IF NOT bOpenClose THEN
	eOpClCtrl := eCtrl;
	THIS^.bCloseWithPiece := bCloseWithPiece;
	fbList.A_AddHeadValue(hList := hList, putValue:= E_Action.ACTION_OpenClose);
	bOpenClose := TRUE;
ELSE
	RETURN;
END_IF

bBusy := TRUE;
eCurrentState := E_MachineState.MACHINESTATE_Active;
END_METHOD

METHOD M_SetAllProps : ERRORID
VAR_INPUT
	refCmdData : REFERENCE TO  ST_CmdData;
END_VAR

VAR
	
END_VAR
M_SetAllProps := SUPER^.M_SetAllProps(refCmdData);

IF M_SetAllProps > 0 THEN
	RETURN;
END_IF

pGripperRef := ADR(pFbMultiZ^.aFbGripperRef[pZAxisRef^.nChannel]);
pZAxisRef^.eFixedToolType := E_MzToolType.TOOL_TYPE_Gripper;
END_METHOD

PROPERTY P_bVialDetector : BOOL
GET
P_bVialDetector :=  pGripperRef^.P_bVialDetector;
END_GET
END_PROPERTY

PROPERTY P_eCurrentGripperState : E_GripperState
GET
P_eCurrentGripperState := pGripperRef^.P_eGripperState;
END_GET
END_PROPERTY

END_FUNCTION_BLOCK

// ---- Objects/Targets/Active/FB_PowderStation.TcPOU
FUNCTION_BLOCK FB_PowderStation EXTENDS FB_ActiveTarget IMPLEMENTS I_SlotTarget
VAR
	
	nNoOfSpecPoints 	: USINT;
	stPickPoint			: ST_3DPoint;
	nLevelOffset		: DINT;
	
	nNoOfSlots			: USINT;
	fbVialSlot			: FB_PieceSlot(pOwner:= THIS);


	//Hardware-Verküpfung
	pPowdStatRef		: POINTER TO FB_HwRefPowderStat;
	
	//Variablen allgemeine Statemachine
	fbSdoWrite			: FB_SDO_WRITE;
	
	//****************************************Aktionvariablen****************************************************
	bActionLock			: ARRAY[50..150] OF BOOL;

	//Action: "Shaking"	(Rüttelmotor schalten)
	bShaking			: BOOL;
	nStateA_Shaking		: USINT;
	nVibrationPower1	: UINT;
	nVibrationPower2	: UINT;
	nVibrationPower3	: UINT;

	//Action: "Leveling"	(Pulver rütteln und auf Höhe bringen)
	bLeveling			: BOOL;				//Action A_Leveling() aktiv setzen
	nStateA_Leveling	: USINT;			//State von A_Leveling()
	tShakingTime		: TIME;
	timer				: TON;
	
	//Action: "Reload"	(Stößel in untere Position fahren zum nachfüllen)
	bReload				: BOOL;
	nStateA_Reload		: USINT;
	
	//Action: "TakePicture"
	bTakePicture			: BOOL;
	nStateA_TakePicture		: USINT;
	tDelayTakePicture		: TIME;
	timerTakePicture		: TON;
	nRequestArg1			: DINT;
	nRequestArg2			: DINT;	
	
END_VAR

IF bInitFB THEN
	bInitFB := FALSE;
	F_CreateLinkedListHnd( ADR( aNodes ), SIZEOF( aNodes ), hList );
	//Fehlerstruktur vorausfüllen
	stError.ObjectId := nObjectID;
	stError.HardwareGrp := E_HardwareGrp.Nothing;
	stError.POU := E_POU.POU_FB_PowderStation;
END_IF

CASE eCurrentState OF
	E_MachineState.MACHINESTATE_Active:
		//BasicActions ausführen
		IF bInit THEN	//Initialisieren
			A_Init();
			IF nStateA_Init >= 80 THEN
				IF nStateA_Init >= 99 THEN
					bError := TRUE;
				END_IF
				bInit := FALSE;
				nStateA_Init := 0;
				M_RemoveListEntry(nSearchValue:= E_Action.ACTION_Init);
			END_IF
		END_IF

		IF bShaking THEN
			A_Shaking();
			IF nStateA_Shaking >= 80 THEN
				IF nStateA_Shaking >= 99 THEN
					bError := TRUE;
				END_IF
				bShaking := FALSE;
				nStateA_Shaking := 0;
				M_RemoveListEntry(nSearchValue:= E_Action.ACTION_PowdStatShaking);
			END_IF
		END_IF
		
		IF bLeveling THEN
			A_Leveling();
			IF nStateA_Leveling >= 80 THEN
				IF nStateA_Leveling >= 99 THEN
					bError := TRUE;
				END_IF
				bLeveling := FALSE;
				nStateA_Leveling := 0;
				M_RemoveListEntry(nSearchValue:= E_Action.ACTION_PowdStatLeveling);
			END_IF
		END_IF
		
		IF bReload THEN
			A_Reload();
			IF nStateA_Reload >= 80 THEN
				IF nStateA_Reload >= 99 THEN
					bError := TRUE;	
				END_IF
				bReload := FALSE;
				nStateA_Reload := 0;
				M_RemoveListEntry(nSearchValue:= E_Action.ACTION_PowdStatReload);
			END_IF
		END_IF

		IF bTakePicture THEN
			A_TakePicture();
			IF nStateA_TakePicture >= 80 THEN
				IF nStateA_TakePicture >= 99 THEN
					bError := TRUE;	
				END_IF
				bTakePicture := FALSE;
				nStateA_TakePicture := 0;
				M_RemoveListEntry(nSearchValue:= E_Action.ACTION_TakePicture);
			END_IF
		END_IF		
		
		IF bStop THEN	//alle Actions stoppen
			A_Stop();
			IF nStateA_Stop >= 80 THEN
				IF nStateA_Stop >= 99 THEN
					bError := TRUE;
				END_IF
				bStop := FALSE;
				nStateA_Stop := 0;
				bCanceled := TRUE;
				M_RemoveListEntry(nSearchValue:= E_Action.ACTION_Stop);
			END_IF							
		END_IF

		IF hList.nCount = 0 THEN
			eCurrentState := E_MachineState.MACHINESTATE_Ready;
		END_IF

		IF bError  THEN
			eCurrentState := E_MachineState.MACHINESTATE_Error;
		END_IF

	E_MachineState.MACHINESTATE_Reset:
		A_Reset();
		IF nStateA_Reset = 80 THEN
			nStateA_Init := 0;
			nStateA_Stop := 0;
			nStateA_Reset := 0;
			bBusy := FALSE;
			bError := FALSE;
			bStopAllOnError := FALSE;
			fbList.A_Reset( hList := hList);
			MEMSET(ADR(bActionLock),0,SIZEOF(bActionLock));
			nErrorId := 0;
			stError.Cmd := 0;
			stError.ErrorId := 0;
			eCurrentState := E_MachineState.MACHINESTATE_Idle;
		ELSIF
			nStateA_Reset = 99 THEN
			fbErrorList.M_Add(stError);
			nStateA_Reset := 0;
			bBusy := FALSE;
			bError := TRUE;
			eCurrentState := E_MachineState.MACHINESTATE_Error;			
		END_IF
	
	E_MachineState.MACHINESTATE_Ready:
		bBusy := FALSE;
		eCurrentState := E_MachineState.MACHINESTATE_Idle;
	
	E_MachineState.MACHINESTATE_Error:
		bBusy := FALSE;
END_CASE

//Prozessdaten aktualisieren
stProcessData.nObjId := nObjectID;
stProcessData.n32Data[0] := BOOL_TO_DINT(bIsInit);
stProcessData.n32Data[1] := eCurrentState;
stProcessData.n32Data[2] := stError.ErrorId;
stProcessData.n32Data[3] := BOOL_TO_DINT(pPowdStatRef^.bLevelOk);	
stProcessData.n32Data[4] := BOOL_TO_DINT(pPowdStatRef^.bLevelLow);
stProcessData.n32Data[5] := BOOL_TO_DINT(pPowdStatRef^.bOnReloadPos);
stProcessData.n32Data[6] := BOOL_TO_DINT(pPowdStatRef^.bVibrationIsOn);
//stProcessData.n32Data[7] := BOOL_TO_DINT(pPowdStatRef^.bCoverIsClosed);
stProcessData.n32Data[7] := BOOL_TO_DINT(pPowdStatRef^.bVialSensor);
stProcessData.n32Data[8] := BOOL_TO_DINT(pPowdStatRef^.bLevelSensor);
stProcessData.n32Data[9] := BOOL_TO_DINT(pPowdStatRef^.bHeaterIsOn);

stProcessData.n32Data[10] := pPowdStatRef^.nTempActual;
IF pPowdStatRef^.P_nCameraLight > 0 THEN
	stProcessData.n32Data[11] := 1;
ELSE
	stProcessData.n32Data[11] := 0;
END_IF
aObjProcData[nNotifyId] := stProcessData;

ACTION A_Init:
CASE nStateA_Init OF
	0:	//Wenn in Error, dann Error zurücksetzen
		bIsInit := FALSE;
		pPowdStatRef^.P_bStartLeveling := FALSE;
		pPowdStatRef^.P_bStartReload := FALSE;
		pPowdStatRef^.P_bVibrationOn := FALSE;
		IF pPowdStatRef^.bErr THEN
			pPowdStatRef^.P_bResetError := TRUE;
			nStateA_Init := 1;
		ELSE
			nStateA_Init := 2;
		END_IF

	1:	//Warten bis Error zurückgesetzt	
		IF NOT pPowdStatRef^.bErr THEN
			pPowdStatRef^.P_bResetError := FALSE;
			nStateA_Init := 2;
		END_IF
		
	2:	//Stöße in ReladPos fahren, wenn noch nicht geschehen
		IF NOT pPowdStatRef^.bOnReloadPos THEN
			pPowdStatRef^.P_bStartReload := TRUE;
			nStateA_Init := 3;
		ELSE
			nStateA_Init := 80;
			bIsInit := TRUE;
		END_IF
	
	3:	//Warten bis Stößel in ReloadPos
		IF pPowdStatRef^.bOnReloadPos THEN
			pPowdStatRef^.P_bStartReload := FALSE;
			nStateA_Init := 80;
			bIsInit := TRUE;	
		END_IF
		IF pPowdStatRef^.bError THEN
			stError.ErrorId := E_ErrorIdCmd.ERRORID_DeviceInErrorState;
			stError.POUState := nStateA_Init;
			nStateA_Init := 99;		
		END_IF
	
	70:	//Initialisierung abbrechen
		pPowdStatRef^.P_bResetError := FALSE;	
		pPowdStatRef^.P_bStartReload := FALSE;
		nStateA_Init := 80;
	
END_CASE

//Errorhandling
IF nStateA_Init = 99 THEN
	stError.Cmd := E_Action.ACTION_Init;
	stError.POUAction := E_POUACT.POUACT_A_Init;
	fbErrorList.M_Add(stError);
END_IF
END_ACTION

ACTION A_Leveling:
stError.POUState := nStateA_Leveling;

IF pPowdStatRef^.bError THEN
	stError.ErrorId := pPowdStatRef^.nError;
	nStateA_Leveling := 99;
	pPowdStatRef^.P_bVibrationOn := FALSE;
END_IF

CASE nStateA_Leveling OF
	0:	//LevelOffset schreiben
		fbSdoWrite(sAdsNetID:= pPowdStatRef^.P_sAdsNetId, nPortNr:= pPowdStatRef^.P_nAdsPort, nIndex:= 16#2104,
					nSubIndex:= 0, nDataLength:= 2, nData:= ABS(nLevelOffset), bExecute:= TRUE);
		IF NOT fbSdoWrite.bBusy THEN
			IF fbSdoWrite.bError THEN
				stError.ErrorId := fbSdoWrite.nAdsErrorId;
				nStateA_Leveling := 99;
			ELSE
				pPowdStatRef^.P_bStartReload := TRUE;
				nStateA_Leveling := 1;
			END_IF
			fbSdoWrite(bExecute:= FALSE);
		END_IF

	1:	//OnReloadPos?
		//Timeout
		timer(IN:=TRUE, PT:= T#5S);
		IF timer.Q THEN
			timer(IN:= FALSE);
			stError.ErrorId := E_ErrorIdCmd.ERRORID_TimeOut;
			nStateA_Leveling := 99;
		END_IF
 
		IF pPowdStatRef^.bOnReloadPos THEN
			timer(IN:=FALSE);
			pPowdStatRef^.P_bStartReload := FALSE;
			IF pPowdStatRef^.bLevelSensor THEN
				stError.ErrorId := E_ErrorIdCmd.ERRORID_PowdDetectOnReloadPos;
				nStateA_Leveling := 99;				
			ELSE
				//ShakerOn, Start Timer
				pPowdStatRef^.P_bVibrationOn := TRUE;
				timer(IN:=TRUE, PT:= tShakingTime);
				nStateA_Leveling := 2;
			END_IF
		END_IF
		
	2:	//Warten bis Timer abgelaufen
		timer();
		IF timer.Q THEN
			timer(IN:= FALSE);
			pPowdStatRef^.P_bVibrationOn := FALSE;
			pPowdStatRef^.P_bStartLeveling := TRUE;
			nStateA_Leveling := 3;
		END_IF
		
	3:	//Warten bis Leveling fertig
		IF pPowdStatRef^.bLevelOk THEN
			pPowdStatRef^.P_bStartLeveling := FALSE;
			nStateA_Leveling := 80;
		ELSIF pPowdStatRef^.bLevelLow THEN
			pPowdStatRef^.P_bStartLeveling := FALSE;
			stError.ErrorId := E_ErrorIdCmd.ERRORID_PowdLevelLow;
			nStateA_Leveling := 99;
		END_IF
		
	70:	//Abbrechen
		pPowdStatRef^.P_bVibrationOn := FALSE;
		pPowdStatRef^.P_bStartLeveling := FALSE;
		pPowdStatRef^.P_bStartReload := FALSE;
		timer(IN:= FALSE);
		nStateA_Leveling := 80;
END_CASE

//Errorhandling
IF nStateA_Leveling = 99 THEN
	stError.Cmd := E_Action.ACTION_PowdStatLeveling;
	stError.POUAction := E_POUACT.POUACT_A_Leveling;
	fbErrorList.M_Add(stError);
END_IF
END_ACTION

ACTION A_Reload:
IF pPowdStatRef^.nError > 0 OR pPowdStatRef^.bError THEN
	stError.POUState := nStateA_Reload;
	stError.ErrorId := pPowdStatRef^.nError;
	nStateA_Reload := 99;
END_IF

CASE nStateA_Reload OF
	0:
		pPowdStatRef^.P_bStartReload := TRUE;
		nStateA_Reload := 1;
		
	1:	//Warten bis Stößel in ReloadPos
		IF pPowdStatRef^.bOnReloadPos THEN
			pPowdStatRef^.P_bStartReload := FALSE;
			nStateA_Reload := 80;
		END_IF
		
	70:	//Abbrechen
		pPowdStatRef^.P_bStartReload := FALSE;
		nStateA_Reload := 80;
END_CASE

//Errorhandling
IF nStateA_Reload = 99 THEN
	stError.Cmd := E_Action.ACTION_PowdStatShaking;
	stError.POUAction := E_POUACT.POUACT_A_Shaking;
	fbErrorList.M_Add(stError);
END_IF
END_ACTION

ACTION A_Reset:
CASE nStateA_Reset OF
	0:
		nStateA_Reset := 80;
END_CASE
END_ACTION

ACTION A_Shaking:
CASE nStateA_Shaking OF
	0:	
		pPowdStatRef^.P_bVibrationOn := TRUE;
		IF tShakingTime > T#0MS THEN
			timer(IN:= TRUE, PT:= tShakingTime);
			nStateA_Shaking := 1;
		END_IF
	1:
		timer();
		IF timer.Q THEN
			pPowdStatRef^.P_bVibrationOn := FALSE;
			timer(IN:= FALSE);
			nStateA_Shaking := 80;
		END_IF
		
	70:	//Abrechen
		pPowdStatRef^.P_bVibrationOn := FALSE;
		timer(IN:=FALSE);
		nStateA_Shaking := 80;
END_CASE
END_ACTION

ACTION A_Stop:
CASE nStateA_Stop OF
	0:
		IF nStateA_Init < 70 AND bInit THEN	//Initialisieren abbrechen
			nStateA_Init := 70;
			nStateA_Stop := 1;	
		END_IF
		
		IF nStateA_Leveling < 70 AND bLeveling THEN
			nStateA_Leveling := 70;
			nStateA_Stop := 1;
		END_IF
		
		IF nStateA_Shaking < 70 AND bShaking THEN
			nStateA_Shaking := 70;
			nStateA_Stop := 1;
		END_IF
		
		IF nStateA_Reload < 70 AND bReload THEN
			nStateA_Reload := 70;
			nStateA_Stop := 1;
		END_IF

	1:	//Warten bis alle Actions fertig abgebrochen
		IF hList.nCount = 1 THEN	//nur der Eintrag von Stop
			nStateA_Stop := 80;
		END_IF
END_CASE
END_ACTION

ACTION A_TakePicture:
IF nStateA_TakePicture = 0 THEN //Timer starten
	timerTakePicture(IN:= TRUE, PT:= tDelayTakePicture);
	IF timerTakePicture.Q THEN
		timerTakePicture(IN:= FALSE);
		stInterResponse.eInteractMessageType := E_InteractMessageType.INTERACTMES_NONE;
		stInteractRequest.eInteractMessageType := E_InteractMessageType.INTERACTMES_WaitForUser;
		stInteractRequest.nObjectId := nObjectID;
		stInteractRequest.nArg1 := nRequestArg1;
		stInteractRequest.nArg2 := nRequestArg2;
		nStateA_TakePicture := 1;
	END_IF
ELSIF nStateA_TakePicture = 1 THEN //Auf InteractResponse warten
	IF stInterResponse.eInteractMessageType = E_InteractMessageType.INTERACTMES_Continue OR 
							stInterResponse.eInteractMessageType = E_InteractMessageType.INTERACTMES_Cancel THEN
		stInteractRequest.eInteractMessageType := E_InteractMessageType.INTERACTMES_NONE;
		nStateA_TakePicture := 80;
	END_IF
ELSIF nStateA_TakePicture = 70 THEN //Abbrechen
	timerTakePicture(IN:= FALSE);
	stInteractRequest.eInteractMessageType := E_InteractMessageType.INTERACTMES_NONE;
	nStateA_TakePicture := 80;
END_IF
END_ACTION

METHOD FB_init : BOOL
VAR_INPUT
	bInitRetains : BOOL; // if TRUE, the retain variables are initialized (warm start / cold start)
	bInCopyCode : BOOL;  // if TRUE, the instance afterwards gets moved into the copy code (online change)
END_VAR
eObjectType := E_ObjectType.OBJECTTYPE_PowderStation;
eObjectGroup := E_ObjectGroup.OBJECTGROUP_Target OR E_ObjectGroup.OBJECTGROUP_Device;
END_METHOD

METHOD M_AddChild : ERRORID
VAR_INPUT
	pObject : POINTER TO FB_Object;
	nSlotNr	: UINT;
	nIndex 	: INT;	
END_VAR
IF pObject > 0 THEN
	IF nSlotNr = fbVialSlot.P_nNr THEN //Reactor besitzt nur den VialSlot
		IF fbVialSlot.P_pChild = 0 THEN
			//Object darf selber noch an keinem Parent hängen
			IF pObject^.P_pParentObject = 0 THEN
				fbVialSlot.P_pChild := pObject;
				pObject^.P_pObjCollectNode := pObjCollectNode^.nodes.M_AddNewNode(pObject,nIndex);
				pObject^.M_UpdateParent();
			ELSE
				M_AddChild := E_ErrorIdObjMgmt.ERRORID_ObjectAlreadyOnAnotherParent;
			END_IF
		ELSE //Slot bereits belegt
			M_AddChild := E_ErrorIdObjMgmt.ERRORID_SlotIsAlreadyOccupied;
		END_IF		
	ELSE
		M_AddChild := SUPER^.M_AddChild(pObject,nSlotNr,nIndex);
	END_IF
ELSE
	M_AddChild := E_ErrorIdObjMgmt.ERRORID_InvalidParentObject;
END_IF
END_METHOD

METHOD M_ApplyPos : ERRORID
VAR_INPUT
	eTargetRef 		: E_TargetRef;
	nPointSlotNr	: UINT;
	stPos 			: ST_3DPoint;
	bXPos			: BOOL;
	bYPos			: BOOL;
	bZPos			: BOOL;	
END_VAR

VAR
	stAbsPos		: ST_3DPoint;
END_VAR
IF eTargetRef = E_TargetRef.TARGETREF_SpecPoint THEN
	IF nPointSlotNr = 1 THEN
		stAbsPos := P_stAbsPosLB;
		IF bXPos THEN
			stPickPoint.X := stPos.X - stAbsPos.X;	
		END_IF
		IF bYPos THEN
			stPickPoint.Y := stPos.Y - stAbsPos.Y;	
		END_IF
		IF bZPos THEN
			stPickPoint.Z := stPos.Z - stAbsPos.Z;	
		END_IF
	ELSE
		M_ApplyPos := E_ErrorIdCmd.ERRORID_InvalidTargetPointNr;
	END_IF
ELSE
	M_ApplyPos := SUPER^.M_ApplyPos(eTargetRef, nPointSlotNr, stPos,bXPos,bYPos,bZPos);
END_IF
END_METHOD

METHOD M_CancelAction
VAR_INPUT
	eAction : E_Action;
END_VAR
CASE eAction OF
	E_Action.ACTION_PowdStatLeveling:
		IF bLeveling AND nStateA_Leveling < 70 THEN
			nStateA_Leveling := 70;
		END_IF
	E_Action.ACTION_PowdStatReload:
		IF bReload AND nStateA_Reload < 70 THEN
			nStateA_Reload := 70;
		END_IF	
	E_Action.ACTION_PowdStatShaking:
		IF bShaking AND nStateA_Shaking < 70 THEN
			nStateA_Shaking := 70;
		END_IF	
END_CASE
END_METHOD

METHOD M_CheckAction : ERRORID
VAR_INPUT
	refActionData 	: REFERENCE TO ST_ActionData;
	pCorrelObject	: POINTER TO FB_Object;
END_VAR
IF refActionData.eAction = E_Action.ACTION_TeachTarget THEN
	IF NOT DINT_TO_UINT(refActionData.aParams[1]) = E_TargetRef.TARGETREF_SpecPoint AND refActionData.aParams[2] = 1 THEN
		M_CheckAction := E_ErrorIdCmd.ERRORID_InvalidTargetPointRef;
	END_IF
END_IF
END_METHOD

METHOD M_CheckProcDataType : BOOL
VAR_INPUT
	eProcDataType : E_ProcDataType;
END_VAR
END_METHOD

METHOD M_ClearAllProps
VAR_INPUT
	bIgnoreParent : BOOL; //Es wird das gesamte OD gelöscht. -> Zeiger auf Parent nicht mehr gültig!
END_VAR
SUPER^.M_ClearAllProps(bIgnoreParent);
fbVialSlot.P_pPiece := 0;
END_METHOD

METHOD M_ExeAction : ERRORID
VAR_INPUT
	refActionData	: REFERENCE TO ST_ActionData;
END_VAR
IF NOT (eCurrentState = E_MachineState.MACHINESTATE_Idle OR
	eCurrentState = E_MachineState.MACHINESTATE_Active OR
	eCurrentState = E_MachineState.MACHINESTATE_Ready) THEN
	M_ExeAction := E_ErrorIdCmd.ERRORID_InvalidState;
	RETURN;
END_IF

CASE refActionData.eAction OF
	E_Action.ACTION_Init:
		IF NOT bInit THEN
			IF pPowdStatRef^.P_bNodeEnabled THEN
				bInit := TRUE;
				fbList.A_AddHeadValue(hList := hList, putValue:= E_Action.ACTION_Init);
				bIsInit := FALSE;
			ELSE
				M_ExeAction := E_ErrorIdCan.ERRORID_NodeNotFound;
				RETURN;
			END_IF
		ELSE
			RETURN;
		END_IF
		
	E_Action.ACTION_PowdStatReload:
		IF NOT bReload THEN
			bReload := TRUE;
			fbList.A_AddHeadValue(hList := hList, putValue:= E_Action.ACTION_PowdStatReload);
		END_IF

	E_Action.ACTION_PowdStatShaking:
		//Aktion wird direkt hier ausgeführt, da in einem Zyklus ausführbar
		IF NOT bIsInit THEN
			M_ExeAction := E_ErrorIdCmd.ERRORID_DeviceNotInitialized;
			RETURN;
		END_IF
		tShakingTime := DINT_TO_TIME(refActionData.aParams[2]);
		nVibrationPower1 := DINT_TO_UINT(refActionData.aParams[3]);
		nVibrationPower2 := DINT_TO_UINT(refActionData.aParams[4]);
		nVibrationPower3 := DINT_TO_UINT(refActionData.aParams[5]);
		
		IF bShaking THEN //Falls Shaker schon Ein
			//Erneuter Einschaltbefehl -> Timer neu setzen
			IF refActionData.aParams[1] = 1 THEN
				timer(IN:= FALSE);
				timer(IN:= TRUE, PT:= tShakingTime);
			ELSE
				nStateA_Shaking := 70; //Abbrechen
			END_IF
		ELSE
			IF refActionData.aParams[1] = 1 THEN
				bShaking := TRUE;
				fbList.A_AddHeadValue(hList := hList, putValue:= E_Action.ACTION_PowdStatShaking);
			END_IF
		END_IF
		
	E_Action.ACTION_PowdStatLeveling:
		IF NOT bIsInit THEN
			M_ExeAction := E_ErrorIdCmd.ERRORID_DeviceNotInitialized;
			RETURN;
		END_IF

		IF NOT bLeveling THEN
			tShakingTime := DINT_TO_TIME(refActionData.aParams[1]);
			bLeveling := TRUE;	
			fbList.A_AddHeadValue(hList := hList, putValue:= E_Action.ACTION_PowdStatLeveling);
		ELSE
			RETURN;
		END_IF
		
	E_Action.ACTION_SwitchLight:	//Beleuchtung für die Kamera
		IF DINT_TO_BOOL(refActionData.aParams[1]) THEN
			pPowdStatRef^.P_nCameraLight := 1023;
		ELSE
			pPowdStatRef^.P_nCameraLight := 0;
		END_IF
		RETURN;
		
	E_Action.ACTION_TakePicture:
		IF NOT bTakePicture THEN
			tDelayTakePicture := DINT_TO_TIME(refActionData.aParams[1]);
			nRequestArg1 := refActionData.aParams[2];
			nRequestArg2 := refActionData.aParams[3];
			bTakePicture := TRUE;
			fbList.A_AddHeadValue(hList := hList, putValue:= E_Action.ACTION_TakePicture);
		ELSE
			RETURN;
		END_IF	
		
	E_Action.ACTION_Stop:
		//Stop braucht nur ausgeführt werden, wenn irgendwas aktiv ist
		IF bBusy AND nStateA_Stop = 0 AND hList.nCount > 0 THEN
			bStop := TRUE;
			fbList.A_AddHeadValue(hList := hList, putValue := E_Action.ACTION_Stop);
		ELSE
			RETURN;
		END_IF
	ELSE
		M_ExeAction := E_ErrorIdCmd.ERRORID_InvalidAction;
END_CASE

bBusy := TRUE;
eCurrentState := E_MachineState.MACHINESTATE_Active;
END_METHOD

METHOD M_GetAbsPos : ST_3DPoint
VAR_INPUT
	pChildPos	: POINTER TO ST_3DPoint;
	eTargetRef 	: E_TargetRef;
	nParam1		: UINT;
 	nParam2		: UINT;
	nParam3		: USINT;
	nParam4		: USINT;
	nZLevel		: USINT;
END_VAR
VAR_OUTPUT
	nErrorId 	: ERRORID;
	lrAngle		: LREAL;
END_VAR
VAR
	stLocPosLB : ST_3DPoint;
END_VAR
IF eTargetRef = E_TargetRef.TARGETREF_SpecPoint THEN
	IF nParam1 = 1 THEN	//Pickpoint X
		stLocPosLB := P_stRelPosLB;
		stLocPosLB := F_Add3DPoints(stLocPosLB,stPickPoint);
		M_GetAbsPos := pParentTarget^.M_GetAbsPos(pChildPos := ADR(stLocPosLB), eTargetRef:= E_TargetRef.TARGETREF_LeftBottom,
													nParam1:= 0,
													nParam2:= 0, nParam3:= 0, nParam4:= 0, nZLevel:= 0,
													lrAngle => lrAngle, nErrorId=> nErrorId);		
	ELSE
		nErrorId := E_ErrorIdCmd.ERRORID_InvalidTargetPointNr;
	END_IF
ELSIF eTargetRef = E_TargetRef.TARGETREF_Slot THEN
	IF nParam1 = 1 THEN
		stLocPosLB := P_stRelPosLB;
		//Slot belegt?
		IF fbVialSlot.P_pPiece > 0 THEN
			stLocPosLB := F_Add3DPoints(stLocPosLB, fbVialSlot.P_pPiece^.M_GetRelPosTopCenter());
		ELSE
			stLocPosLB := F_Add3DPoints(stLocPosLB,fbVialSlot.P_stRelPos);	
		END_IF
		
		M_GetAbsPos := pParentTarget^.M_GetAbsPos(pChildPos := ADR(stLocPosLB), eTargetRef:= E_TargetRef.TARGETREF_LeftBottom,
													nParam1:= 0,
													nParam2:= 0, nParam3:= 0, nParam4:= 0, nZLevel:= 0,
													lrAngle => lrAngle, nErrorId=> nErrorId);		
	ELSE
		nErrorId := E_ErrorIdCmd.ERRORID_InvalidTargetPointNr;
	END_IF	
ELSE
	M_GetAbsPos := SUPER^.M_GetAbsPos(pChildPos := pChildPos, eTargetRef:= eTargetRef,
													nParam1:= nParam1,
													nParam2:= nParam2, nParam3:= nParam3, nParam4:= 0, nZLevel:= nZLevel,
													lrAngle => lrAngle, nErrorId=> nErrorId);		
END_IF
END_METHOD

METHOD M_GetActionBusy : BOOL
VAR_INPUT
	eAction : E_Action;
END_VAR
getPosPtr := 0;(* start from first node element *)
fbList.A_FindNext( hList := hList, putPosPtr := getPosPtr, putValue := eAction, getValue=>getValue, getPosPtr=>getPosPtr );
IF fbList.bOk THEN	//Eintrag wurde gefunden, d.h. Action ist noch busy
	M_GetActionBusy := TRUE;
END_IF
END_METHOD

METHOD M_GetAllProps : ERRORID
VAR_INPUT
	refCmdData : REFERENCE TO  ST_CmdData;
END_VAR
SUPER^.M_GetAllProps(refCmdData);

nCurrentPropIndex := nCurrentPropIndex + 1;
refCmdData.n32Data[nCurrentPropIndex] := nNoOfSlots;
nCurrentPropIndex := nCurrentPropIndex + 1;
refCmdData.n32Data[nCurrentPropIndex] := fbVialSlot.nNr;
nCurrentPropIndex := nCurrentPropIndex + 1;
refCmdData.n32Data[nCurrentPropIndex] := REAL_TO_DINT(fbVialSlot.P_rRelPosX);
nCurrentPropIndex := nCurrentPropIndex + 1;
refCmdData.n32Data[nCurrentPropIndex] := REAL_TO_DINT(fbVialSlot.P_rRelPosY);
nCurrentPropIndex := nCurrentPropIndex + 1;
refCmdData.n32Data[nCurrentPropIndex] := REAL_TO_DINT(fbVialSlot.P_rRelPosZ);
nCurrentPropIndex := nCurrentPropIndex + 1;
refCmdData.n32Data[nCurrentPropIndex] := REAL_TO_DINT(fbVialSlot.P_rDepth);

nCurrentPropIndex := nCurrentPropIndex + 1;
refCmdData.n32Data[nCurrentPropIndex] := nNoOfSpecPoints;
nCurrentPropIndex := nCurrentPropIndex + 1;
refCmdData.n32Data[nCurrentPropIndex] := REAL_TO_DINT(stPickPoint.X);
nCurrentPropIndex := nCurrentPropIndex + 1;
refCmdData.n32Data[nCurrentPropIndex] := REAL_TO_DINT(stPickPoint.Y);
nCurrentPropIndex := nCurrentPropIndex + 1;
refCmdData.n32Data[nCurrentPropIndex] := REAL_TO_DINT(stPickPoint.Z);
nCurrentPropIndex := nCurrentPropIndex + 1;
refCmdData.n32Data[nCurrentPropIndex] := pPowdStatRef^.nPidKp;
nCurrentPropIndex := nCurrentPropIndex + 1;
refCmdData.n32Data[nCurrentPropIndex] := pPowdStatRef^.nPidKi;
nCurrentPropIndex := nCurrentPropIndex + 1;
refCmdData.n32Data[nCurrentPropIndex] := pPowdStatRef^.nPidKd;
nCurrentPropIndex := nCurrentPropIndex + 1;
refCmdData.n32Data[nCurrentPropIndex] := pPowdStatRef^.nPidTa;
nCurrentPropIndex := nCurrentPropIndex + 1;
refCmdData.n32Data[nCurrentPropIndex] := pPowdStatRef^.nVibrationPower1;
nCurrentPropIndex := nCurrentPropIndex + 1;
refCmdData.n32Data[nCurrentPropIndex] := pPowdStatRef^.nVibrationPower2;
nCurrentPropIndex := nCurrentPropIndex + 1;
refCmdData.n32Data[nCurrentPropIndex] := pPowdStatRef^.nVibrationPower3;
nCurrentPropIndex := nCurrentPropIndex + 1;
refCmdData.n32Data[nCurrentPropIndex] := nLevelOffset;
END_METHOD

METHOD M_GetProcData : DINT
VAR_INPUT
	eProcDataType : E_ProcDataType;
END_VAR
END_METHOD

METHOD M_GetSlot : POINTER TO FB_Slot
VAR_INPUT
	nSlotNr : UINT;
END_VAR
IF nSlotNr = 1 THEN
	M_GetSlot := ADR(fbVialSlot);
END_IF
END_METHOD

METHOD M_GetSlotFromChild : POINTER TO FB_Slot
VAR_INPUT
	pObject : POINTER TO FB_Object;
END_VAR
IF fbVialSlot.P_pChild = pObject THEN
	M_GetSlotFromChild := ADR(fbVialSlot);
END_IF
END_METHOD

METHOD M_RemoveListEntry : BOOL
VAR_INPUT
	nSearchValue : E_Action;
END_VAR
getPosPtr := 0;(* start from first node element *)
fbList.A_FindNext( hList := hList, putPosPtr := getPosPtr, putValue := nSearchValue, getValue=>getValue, getPosPtr=>getPosPtr );
IF fbList.bOk THEN	//Eintrag wurde gefunden
	fbList.A_RemoveValueAtPosPtr(hList:= hList,	putPosPtr:= getPosPtr);
	IF fbList.bOk THEN
		M_RemoveListEntry := TRUE;
	END_IF
END_IF
END_METHOD

METHOD M_SetAllProps : ERRORID
VAR_INPUT
	refCmdData : REFERENCE TO  ST_CmdData;
END_VAR
M_SetAllProps := SUPER^.M_SetAllProps(refCmdData);

IF M_SetAllProps > 0 THEN
	RETURN;
END_IF

nCurrentPropIndex := nCurrentPropIndex + 1;
nSpecPropIndex := nCurrentPropIndex;
//NumberOfSlots immer "1"
nNoOfSlots := DINT_TO_USINT(refCmdData.n32Data[nCurrentPropIndex]);
IF nNoOfSlots <> 1 THEN
	nNoOfSlots := 1;
	M_SetAllProps := E_ErrorIdObjMgmt.ERRORID_InvalidNoOfSlots;
	RETURN;
END_IF
nCurrentPropIndex := nCurrentPropIndex + 1;
fbVialSlot.P_nNr := DINT_TO_UINT(refCmdData.n32Data[nCurrentPropIndex]);
//SlotNr immer "1"
IF fbVialSlot.P_nNr <> 1 THEN
	fbVialSlot.P_nNr := 1;
	M_SetAllProps := E_ErrorIdObjMgmt.ERRORID_InvalidSlotNumber;
	RETURN;
END_IF

nCurrentPropIndex := nCurrentPropIndex + 1;
fbVialSlot.P_rRelPosX := DINT_TO_REAL(refCmdData.n32Data[nCurrentPropIndex]);
nCurrentPropIndex := nCurrentPropIndex + 1;
fbVialSlot.P_rRelPosY := DINT_TO_REAL(refCmdData.n32Data[nCurrentPropIndex]);
nCurrentPropIndex := nCurrentPropIndex + 1;
fbVialSlot.P_rRelPosZ := DINT_TO_REAL(refCmdData.n32Data[nCurrentPropIndex]);
nCurrentPropIndex := nCurrentPropIndex + 1;
fbVialSlot.P_rDepth := DINT_TO_REAL(refCmdData.n32Data[nCurrentPropIndex]);

{IF defined (variable:aFbPowderStatRef)}
nCurrentPropIndex := nCurrentPropIndex + 1;
nSpecPropIndex := nCurrentPropIndex;
nNoOfSpecPoints := DINT_TO_USINT(refCmdData.n32Data[nCurrentPropIndex]);
nCurrentPropIndex := nCurrentPropIndex + 1;
stPickPoint.X := DINT_TO_REAL(refCmdData.n32Data[nCurrentPropIndex]);
nCurrentPropIndex := nCurrentPropIndex + 1;
stPickPoint.Y := DINT_TO_REAL(refCmdData.n32Data[nCurrentPropIndex]);
nCurrentPropIndex := nCurrentPropIndex + 1;
stPickPoint.Z := DINT_TO_REAL(refCmdData.n32Data[nCurrentPropIndex]);
nCurrentPropIndex := nCurrentPropIndex + 1;
pPowdStatRef := ADR(aFbPowderStatRef[1]);
pPowdStatRef^.P_nPidKp := DINT_TO_UINT(refCmdData.n32Data[nCurrentPropIndex]);
nCurrentPropIndex := nCurrentPropIndex + 1;
pPowdStatRef^.P_nPidKi := DINT_TO_UINT(refCmdData.n32Data[nCurrentPropIndex]);
nCurrentPropIndex := nCurrentPropIndex + 1;
pPowdStatRef^.P_nPidKd := DINT_TO_UINT(refCmdData.n32Data[nCurrentPropIndex]);
nCurrentPropIndex := nCurrentPropIndex + 1;
pPowdStatRef^.P_nPidTa := DINT_TO_USINT(refCmdData.n32Data[nCurrentPropIndex]);
nCurrentPropIndex := nCurrentPropIndex + 1;
pPowdStatRef^.P_nVibrationPower1 := DINT_TO_UINT(refCmdData.n32Data[nCurrentPropIndex]);
nCurrentPropIndex := nCurrentPropIndex + 1;
pPowdStatRef^.P_nVibrationPower2 := DINT_TO_UINT(refCmdData.n32Data[nCurrentPropIndex]);
nCurrentPropIndex := nCurrentPropIndex + 1;
pPowdStatRef^.P_nVibrationPower3 := DINT_TO_UINT(refCmdData.n32Data[nCurrentPropIndex]);
{ELSE}
M_SetAllProps := E_ErrorIdObjMgmt.ERRORID_InvalidHardwareRef;
RETURN;
{END_IF}
nCurrentPropIndex := nCurrentPropIndex + 1;
nLevelOffset := refCmdData.n32Data[nCurrentPropIndex];
nNoOfProps := nCurrentPropIndex + 1;
END_METHOD

METHOD M_SetSingleProp : ERRORID
VAR_INPUT
	refCmdData : REFERENCE TO  ST_CmdData;
END_VAR
IF nSpecPropIndex = refCmdData.aHeader[1] THEN
	M_SetSingleProp := E_ErrorIdCmd.ERRORID_InvalidProperty; //Anzahl Specpoints darf nicht verändert werden
ELSIF (nSpecPropIndex + 1) = refCmdData.aHeader[1] THEN
	stPickPoint.X := DINT_TO_REAL(refCmdData.n32Data[0]);
ELSIF (nSpecPropIndex + 2) = refCmdData.aHeader[1] THEN
	stPickPoint.Y := DINT_TO_REAL(refCmdData.n32Data[0]);
ELSIF (nSpecPropIndex + 3) = refCmdData.aHeader[1] THEN
	stPickPoint.Z := DINT_TO_REAL(refCmdData.n32Data[0]);
ELSIF (nSpecPropIndex + 4) = refCmdData.aHeader[1] THEN
	pPowdStatRef^.P_nPidKp := DINT_TO_UINT(refCmdData.n32Data[0]);
ELSIF (nSpecPropIndex + 5) = refCmdData.aHeader[1] THEN
	pPowdStatRef^.P_nPidKi := DINT_TO_UINT(refCmdData.n32Data[0]);
ELSIF (nSpecPropIndex + 6) = refCmdData.aHeader[1] THEN
	pPowdStatRef^.P_nPidKd := DINT_TO_UINT(refCmdData.n32Data[0]);
ELSIF (nSpecPropIndex + 7) = refCmdData.aHeader[1] THEN
	pPowdStatRef^.P_nPidTa := DINT_TO_USINT(refCmdData.n32Data[0]);
ELSIF (nSpecPropIndex + 8) = refCmdData.aHeader[1] THEN
	pPowdStatRef^.P_nVibrationPower1 := DINT_TO_UINT(refCmdData.n32Data[0]);
ELSIF (nSpecPropIndex + 9) = refCmdData.aHeader[1] THEN
	pPowdStatRef^.P_nVibrationPower2 := DINT_TO_UINT(refCmdData.n32Data[0]);
ELSIF (nSpecPropIndex + 10) = refCmdData.aHeader[1] THEN
	pPowdStatRef^.P_nVibrationPower3 := DINT_TO_UINT(refCmdData.n32Data[0]);
ELSIF (nSpecPropIndex + 11) = refCmdData.aHeader[1] THEN
	nLevelOffset := refCmdData.n32Data[0];
ELSE
	M_SetSingleProp := SUPER^.M_SetSingleProp(refCmdData);
END_IF
END_METHOD

METHOD PRIVATE M_SetSpeed : BOOL
VAR_INPUT
	nSpeed : UDINT;
END_VAR

VAR_OUTPUT
	nErrorId	: ERRORID;
END_VAR
(*//Profile Speed setzen
fbSdoWrite(sADSNetID:= stPowdStatRef.stAdsAdress.sNetId,nPortNr:= stPowdStatRef.stAdsAdress.nPort, 
			nIndex:= 16#6081, nSubIndex:= 0, nDataLength:= 4, nData:= UDINT_TO_DINT(nSpeed), bExecute:= TRUE);

M_SetSpeed := fbSdoWrite.bBusy; 

IF NOT fbSdoWrite.bBusy THEN
	IF fbSdoWrite.bError THEN
		nErrorId := fbSdoWrite.nAdsErrorId;
	END_IF
	fbSdoWrite(bExecute:= FALSE);
END_IF			
*)
END_METHOD

METHOD M_Stop : ERRORID
VAR_INPUT
END_VAR
//Stop braucht nur ausgeführt werden, wenn irgendwas aktiv ist
IF NOT bStop AND eCurrentState = E_MachineState.MACHINESTATE_Active THEN
 	//stPowdStatRef.bShaker := FALSE;
	bStop := TRUE;
	fbList.A_AddHeadValue(hList := hList, putValue := E_Action.ACTION_Stop);
END_IF
END_METHOD

PROPERTY P_bVialSensor : BOOL
GET
P_bVialSensor := pPowdStatRef^.P_bVialSensor;
END_GET
END_PROPERTY

PROPERTY P_pVial : POINTER TO FB_Vial
GET
P_pVial := fbVialSlot.P_pPiece;
END_GET
SET
fbVialSlot.P_pPiece := P_pVial;
END_SET
END_PROPERTY

END_FUNCTION_BLOCK

// ---- Hardware/PowderStation/FB_HwRefPowderStat.TcPOU
FUNCTION_BLOCK FB_HwRefPowderStat EXTENDS FB_CanNodeBase
VAR_INPUT
END_VAR
VAR_OUTPUT
END_VAR
VAR
	//Eingänge
	nTempActual 	AT %I* : UINT;	//aktuelle Temperatur in 1/100tel °C
	
	//Anfang StatusByte 
	bLevelOk		AT %I* : BOOL;	//Bit0 - Level erreicht
	bOnReloadPos	AT %I* : BOOL;	//Bit1 - Stößel ganz unten
	bHeaterIsOn		AT %I* : BOOL;	//Bit2 - Heizung aktiv
	bVibrationIsOn	AT %I* : BOOL;	//Bit3 - Vibrationmotoren sind ein
	bLevelLow		AT %I* : BOOL;	//Bit4 - Level wurde nicht erreicht 
	//bCoverIsClosed	(*AT %I**) : BOOL := TRUE;	//Bit5 - Deckel ist offen (obsolet für Generation 2)
	bVialSensor		AT %I* : BOOL;	//Bit5 - VialSensor
	bLevelSensor	AT %I* : BOOL;	//Bit6 - LevelSensor
	bErr			AT %I* : BOOL; 	//Bit7 - Error
	//Ende StatusByte
	
	nError			AT %I* : USINT;	//ErrorValue
	
	//Ausgänge
	nPidKp 			AT %Q* : UINT; 	//PID-Reglerparameter KP
	nPidKi 			AT %Q* : UINT;	//PID-Reglerparameter KI
	nPidKd 			AT %Q* : UINT;	//PID-Reglerparameter KD
	nPidTa 			AT %Q* : USINT;	//PID-Reglerparameter TA
	bHeatingOn		AT %Q* : BOOL;	//Heizer EIN
	
	nTempSetpoint	AT %Q* : USINT;	//Solltemperatur in °C (ohne Kommastellen)
	//Anfang ControlByte
	bStartLeveling	AT %Q* : BOOL;	//Bit0 - Start Leveling
	bStartReload	AT %Q* : BOOL;	//Bit1 - Bewege Stöße zu ReloadPos
	bVibrationOn	AT %Q* : BOOL;	//Bit2 - Vibrationsmotoren ein
	bResetErr		AT %Q* : BOOL;	//Bit3 - Error zurücksetzen
	//Ende ControlByte
	
	nVibrationPower1 AT %Q* : UINT;
	nVibrationPower2 AT %Q* : UINT;
	nVibrationPower3 AT %Q* : UINT;	
	
	nCameraLight	AT %Q* : UINT;
END_VAR

IF bNodeEnabled THEN
	SUPER^();	
END_IF

PROPERTY P_bResetError : BOOL
SET
bResetErr := P_bResetError;
END_SET
END_PROPERTY

PROPERTY P_bStartLeveling : BOOL
GET
P_bStartLeveling := bStartLeveling;
END_GET
SET
bStartLeveling := P_bStartLeveling;
END_SET
END_PROPERTY

PROPERTY P_bStartReload : BOOL
GET
P_bStartReload := bStartReload;
END_GET
SET
bStartReload := P_bStartReload;
END_SET
END_PROPERTY

PROPERTY P_bVialSensor : BOOL
GET
P_bVialSensor := bVialSensor;
END_GET
END_PROPERTY

PROPERTY P_bVibrationOn : BOOL
GET
P_bVibrationOn := bVibrationOn;
END_GET
SET
bVibrationOn := P_bVibrationOn;
END_SET
END_PROPERTY

PROPERTY P_nCameraLight : UINT
GET
P_nCameraLight := nCameraLight;
END_GET
SET
nCameraLight := P_nCameraLight;
END_SET
END_PROPERTY

PROPERTY P_nPidKd : UINT
GET
P_nPidKd := nPidKd;
END_GET
SET
nPidKd := P_nPidKd;
END_SET
END_PROPERTY

PROPERTY P_nPidKi : UINT
GET
P_nPidKi := nPidKi;
END_GET
SET
nPidKi := P_nPidKi;
END_SET
END_PROPERTY

PROPERTY P_nPidKp : UINT
GET
P_nPidKp := nPidKp;
END_GET
SET
nPidKp := P_nPidKp;
END_SET
END_PROPERTY

PROPERTY P_nPidTa : USINT
GET
P_nPidTa := nPidTa;
END_GET
SET
nPidTa := P_nPidTa;
END_SET
END_PROPERTY

PROPERTY P_nTempActual : UINT
GET
P_nTempActual := nTempActual;
END_GET
END_PROPERTY

PROPERTY P_nTempSetpoint : USINT
GET
P_nTempSetpoint := nTempSetpoint;
END_GET
SET
nTempSetpoint := P_nTempSetpoint;
END_SET
END_PROPERTY

PROPERTY P_nVibrationPower1 : UINT
GET
P_nVibrationPower1 := nVibrationPower1;
END_GET
SET
nVibrationPower1 := P_nVibrationPower1;
END_SET
END_PROPERTY

PROPERTY P_nVibrationPower2 : UINT
GET
P_nVibrationPower2 := nVibrationPower2;
END_GET
SET
nVibrationPower2 := P_nVibrationPower2;
END_SET
END_PROPERTY

PROPERTY P_nVibrationPower3 : UINT
GET
P_nVibrationPower3 := nVibrationPower3;
END_GET
SET
nVibrationPower3 := P_nVibrationPower3;
END_SET
END_PROPERTY

END_FUNCTION_BLOCK

// ---- Objects/Tools/FB_PickPlacePip.TcPOU
FUNCTION_BLOCK FB_PickPlacePip EXTENDS FB_GCodeTool

VAR

	//Specproperties
	pPneuChannelPress	: POINTER TO FB_PneuChannelRef;
	pPneuChannelVac		: POINTER TO FB_PneuChannelRef;
	
	nValveNrPress		: USINT;	//Druckventil
	nValveNrVac			: USINT;	//Vakuumventil 
	
	//****************************************Aktionvariablen****************************************************
	
	//Action: "InitTool"
	bInitTool			: BOOL;
	nStateA_InitTool	: USINT;	

	//Action: "SetPressure"
	bSetPress			: BOOL;
	fbSetPress			: FB_SetPressure;

	//Action: "SetVacuum"
	bSetVacuum			: BOOL;
	fbSetVacuum			: FB_SetPressure;
	
	//Action: "SwitchPressure"
	bSwitchPress		: BOOL;
	nStateA_SwitchPress	: USINT;	//State von A_SwitchPress()
	ePressCtrl			: E_PressCtrl;
	eCurrPressCtrl 		: E_PressCtrl; 
	tPressTime			: TIME;		//Öffnungszeit Druckventil
	timerPress			: TON;		//Timer für Öffnungszeit Druckventil
	
	//Action: "PulsePressure"
	bPulsePress			: BOOL;
	nStateA_PulsePress	: USINT;	//State von A_PulsePress()
	eSwitchCtrlPhase1	: E_PressCtrl;		//
	eSwitchCtrlPhase2	: E_PressCtrl;		//
	nPulseDutycycle		: UINT;		//Tastverhältnis (0-100%)
	nTimePhase1			: UINT;
	nTimePhase2			: UINT;
	timerPulse			: TON;		//Timer
	nSetpointPulses		: UINT;		//Soll Anzahl an Pulses
	nCurrentPulses		: UINT;		//aktuelle Anzahl an Pulses
	bPulseOn			: BOOL;	
	
	//Action: "PickPut
	bPickPut			: BOOL;
	nStateA_PickPut		: USINT;
	ePickPutMode		: E_PickPutMode;
	nIntakeVac			: INT;
	tIntakeTime			: TIME;
	nHoldVac			: INT;
	nBlowOutPress		: INT;
	nBlowOutPulseTime	: UINT;
	nBlowOutPulses		: UINT;
	timerPickPut		: TON;
	stActionDataPickPut	: ST_ActionData;	
	
END_VAR

IF eCurrentState = E_MachineState.MACHINESTATE_Active THEN
	
	IF bPickPut THEN
		A_PickPut();
		IF nStateA_PickPut >= 80 THEN
			IF nStateA_PickPut >= 99 THEN
				bError := TRUE;
			END_IF
			bPickPut := FALSE;
			nStateA_PickPut := 0;
			M_RemoveListEntry(nSearchValue:= E_Action.ACTION_PickPutPowder);
		END_IF
	END_IF		
	
	IF bSetPress THEN
		fbSetPress(pPneuChannelRef:= pPneuChannelPress);
		IF NOT fbSetPress.bBusy THEN
			IF fbSetPress.bError THEN
				bError := TRUE;
				stError.ErrorId := fbSetPress.nErrorId;
				stError.POU := E_POU.POU_FB_PowderPip;
				fbErrorList.M_Add(stError);
			END_IF
			bSetPress := FALSE;
			fbSetPress(pPneuChannelRef:= pPneuChannelPress, bExecute:= FALSE);
			M_RemoveListEntry(nSearchValue:= E_Action.ACTION_SetPressure);
		END_IF
	END_IF	

	IF bSetVacuum THEN
		fbSetVacuum(pPneuChannelRef:= pPneuChannelVac);
		IF NOT fbSetVacuum.bBusy THEN
			IF fbSetVacuum.bError THEN
				bError := TRUE;
				stError.ErrorId := fbSetVacuum.nErrorId;
				stError.POU := E_POU.POU_FB_PowderPip;
				fbErrorList.M_Add(stError);
			END_IF
			bSetVacuum := FALSE;
			fbSetVacuum(pPneuChannelRef:= pPneuChannelVac, bExecute:= FALSE);
			M_RemoveListEntry(nSearchValue:= E_Action.ACTION_SetVacuum);
		END_IF
	END_IF	

	IF bSwitchPress THEN	//Druck/Vakuum Ein/Aus
		A_SwitchPress();
		IF nStateA_SwitchPress >= 80 THEN
			IF nStateA_SwitchPress >= 99 THEN
				bError := TRUE;
			END_IF
			bSwitchPress := FALSE;
			nStateA_SwitchPress := 0;
			M_RemoveListEntry(nSearchValue:= E_Action.ACTION_SwitchPressure);
		END_IF
	END_IF
	
	IF bPulsePress THEN
		A_PulsePress();
		IF nStateA_PulsePress >= 80 THEN
			IF nStateA_PulsePress >= 99 THEN
				bError := TRUE;
			END_IF
			bPulsePress := FALSE;
			nStateA_PulsePress := 0;
			M_RemoveListEntry(nSearchValue:= E_Action.ACTION_PulsePressure);
		END_IF
	END_IF
END_IF

SUPER^();	//FB_MzTool aufrufen

//Prozessdaten aktualisieren

IF pPneuChannelPress > 0 THEN
	stProcessData.n32Data[7] := pPneuChannelPress^.P_nCurrentPressure;
	stProcessData.n32Data[8] := pPneuChannelPress^.P_nCurrentPressure;
END_IF

IF pPneuChannelVac > 0 THEN
	stProcessData.n32Data[9] := pPneuChannelVac^.P_nSetPressure;
	stProcessData.n32Data[10] := pPneuChannelVac^.P_nCurrentPressure;
END_IF

IF nValveNrPress > 0 AND nValveNrVac > 0 THEN
	IF aValves[nValveNrPress].bDigiOut1 THEN
		stProcessData.n32Data[11] := E_PressCtrl.PRESSCTRL_PressOn;
	ELSIF aValves[nValveNrVac].bDigiOut1 THEN
 		stProcessData.n32Data[11] := E_PressCtrl.PRESSCTRL_VacOn;
	ELSE
		stProcessData.n32Data[11] := E_PressCtrl.PRESSCTRL_Off;
	END_IF
ELSIF nValveNrPress > 0 THEN
	IF aValves[nValveNrPress].bDigiOut1 THEN
		stProcessData.n32Data[11] := E_PressCtrl.PRESSCTRL_PressOn;
	ELSE
		stProcessData.n32Data[11] := E_PressCtrl.PRESSCTRL_Off;
	END_IF
ELSIF nValveNrVac > 0 THEN 
	IF aValves[nValveNrVac].bDigiOut1 THEN
		stProcessData.n32Data[11] := E_PressCtrl.PRESSCTRL_VacOn;
	ELSE
		stProcessData.n32Data[11] := E_PressCtrl.PRESSCTRL_Off;
	END_IF
ELSE
	stProcessData.n32Data[11] := E_PressCtrl.PRESSCTRL_UNDEFINED;
END_IF

aObjProcData[nNotifyId] := stProcessData;

ACTION A_PickPut:
CASE nStateA_PickPut OF
	0:	//Ventile schließen
		pZAxisRef^.stOutput.nToolCtrl := 0;
		//Wenn Pick IntakeVac einstellen, bei Put BlowOutPress einstellen
		MEMSET(ADR(stActionDataPickPut),0,SIZEOF(stActionDataPickPut));
		IF ePickPutMode = E_PickPutMode.MODE_Pick THEN
			stActionDataPickPut.eAction := E_Action.ACTION_SetVacuum;
			stActionDataPickPut.aParams[2] := nIntakeVac;	
		ELSIF ePickPutMode = E_PickPutMode.MODE_Put THEN
			stActionDataPickPut.eAction := E_Action.ACTION_SetPressure;
			stActionDataPickPut.aParams[2] := nBlowOutPress;
			GVL_HwRefIO.bTrigger1 := TRUE;
		END_IF
		stActionDataPickPut.aParams[1] := 1;	//Fertigmeldung erst, wenn Druck erreicht
		stActionDataPickPut.aParams[3] := 8;	//Tolerance +
		stActionDataPickPut.aParams[4] := 8;	//Tolerance -
		stActionDataPickPut.aParams[5] := 10000; //Timeout
		M_ExeAction(stActionDataPickPut);
		stActionDataPickPut.eAction := E_Action.ACTION_SwitchPressure;
		stActionDataPickPut.aParams[1] := E_PressCtrl.PRESSCTRL_Off;
		M_ExeAction(stActionDataPickPut);
		nStateA_PickPut := 1;
	
	1:	//Warten bis SollDruck erreioht ist
		IF NOT M_GetActionBusy(E_Action.ACTION_SetPressure) AND NOT M_GetActionBusy(E_Action.ACTION_SetVacuum)THEN
			IF ePickPutMode = E_PickPutMode.MODE_Pick THEN
				nStateA_PickPut := 2;
			ELSE
				nStateA_PickPut := 20;
			END_IF
		END_IF
		
	2:	//Pick - Switch Vacuum
		MEMSET(ADR(stActionDataPickPut),0,SIZEOF(stActionDataPickPut));
		stActionDataPickPut.eAction := E_Action.ACTION_SwitchPressure;
		stActionDataPickPut.aParams[1] := E_PressCtrl.PRESSCTRL_VacOn;
		stActionDataPickPut.aParams[2] := 0;
		M_ExeAction(stActionDataPickPut);
		timerPickPut(IN:=TRUE, PT:= tIntakeTime);
		nStateA_PickPut := 3;

	3:	//Warten, bis Zeit abgelaufen
		timerPickPut();
		IF timerPickPut.Q THEN
			timerPickPut(IN:= FALSE);
			MEMSET(ADR(stActionDataPickPut),0,SIZEOF(stActionDataPickPut));
			//HoldVac einstellen (wenn HoldVac = 0, dann SwitchPress auf Off
			IF nHoldVac < 0 THEN
				stActionDataPickPut.eAction := E_Action.ACTION_SetVacuum;
				stActionDataPickPut.aParams[1] := 0; //Ohne Überwachung
				stActionDataPickPut.aParams[2] := nHoldVac;
				M_ExeAction(stActionDataPickPut);
			ELSE
				stActionDataPickPut.eAction := E_Action.ACTION_SwitchPressure;
				stActionDataPickPut.aParams[1] := E_PressCtrl.PRESSCTRL_Off;
				stActionDataPickPut.aParams[2] := 0;
				M_ExeAction(stActionDataPickPut);
			END_IF
			nStateA_PickPut := 80;
		END_IF
		
	20:	//Put
		//PulsePressure
		MEMSET(ADR(stActionDataPickPut),0,SIZEOF(stActionDataPickPut));
		stActionDataPickPut.eAction := E_Action.ACTION_PulsePressure;
		stActionDataPickPut.aParams[1] := E_PressCtrl.PRESSCTRL_PressOn;
		stActionDataPickPut.aParams[2] := E_PressCtrl.PRESSCTRL_Off;
		stActionDataPickPut.aParams[3] := nBlowOutPulseTime * 2; //Periode
		stActionDataPickPut.aParams[4] := 50; //Dutycycle
		stActionDataPickPut.aParams[5] := nBlowOutPulses;
		stActionDataPickPut.aParams[6] := 1; //On
		M_ExeAction(stActionDataPickPut);
		nStateA_PickPut := 21;
		
	21: //Warten, bis Pulsen fertig
		IF NOT M_GetActionBusy(E_Action.ACTION_PulsePressure) THEN
			GVL_HwRefIO.bTrigger1 := FALSE;
			nStateA_PickPut := 80;
		END_IF
	
	70: //Abbrechen
		M_CancelAction(E_Action.ACTION_PulsePressure);
		stActionDataPickPut.eAction := E_Action.ACTION_SwitchPressure;
		stActionDataPickPut.aParams[1] := E_PressCtrl.PRESSCTRL_Off;
		M_ExeAction(stActionDataPickPut);
		timerPickPut(IN:= FALSE);
		nStateA_PickPut := 80;
		
END_CASE
END_ACTION

ACTION A_PulsePress:
CASE nStateA_PulsePress OF
	0:	//Phase1
		
		IF eSwitchCtrlPhase1 = E_PressCtrl.PRESSCTRL_Off THEN
			M_PressAndVacOff();
		ELSIF eSwitchCtrlPhase1 = E_PressCtrl.PRESSCTRL_PressOn THEN
			M_PressOn();
		ELSIF eSwitchCtrlPhase1 = E_PressCtrl.PRESSCTRL_VacOn THEN
			M_VacOn();
		END_IF

		timerPulse(IN:= TRUE, PT:= UINT_TO_TIME(nTimePhase1));
		IF timerPulse.Q THEN
			timerPulse(IN:= FALSE);
			nStateA_PulsePress := 1;
			nCurrentPulses := nCurrentPulses + 1;
		END_IF

	1:	//Phase2

		IF eSwitchCtrlPhase2 = E_PressCtrl.PRESSCTRL_Off THEN
			M_PressAndVacOff();
		ELSIF eSwitchCtrlPhase2 = E_PressCtrl.PRESSCTRL_PressOn THEN
			M_PressOn();
		ELSIF eSwitchCtrlPhase2 = E_PressCtrl.PRESSCTRL_VacOn THEN
			M_VacOn();
		END_IF

		timerPulse(IN:= TRUE, PT:= UINT_TO_TIME(nTimePhase2));
		IF timerPulse.Q THEN
			timerPulse(IN:= FALSE);
			IF nCurrentPulses = nSetpointPulses THEN
				M_PressAndVacOff();
				nStateA_PulsePress := 80;
			ELSIF nSetpointPulses = 0 AND NOT bPulseOn THEN
				M_PressAndVacOff();
				nStateA_PulsePress := 80;
			ELSE
				nStateA_PulsePress := 0;	
			END_IF
		END_IF
		
	70:	//Abbrechen
		timerPulse(IN:= FALSE);
		M_PressAndVacOff();
		nStateA_PulsePress := 80;
		
END_CASE
END_ACTION

ACTION A_Reset:
//Ist noch eine Aktion aktiv?
IF nStateA_ResetSpec = 0 THEN 
	IF bSetPress THEN
		bSetPress := FALSE;
		fbSetPress(bExecute:= FALSE, pPneuChannelRef:= pPneuChannelPress);
	END_IF

	IF bSetVacuum THEN
		bSetVacuum := FALSE;
		fbSetVacuum(bExecute:= FALSE, pPneuChannelRef:= pPneuChannelVac);
	END_IF
	
	IF bSwitchPress THEN 
		bSwitchPress := FALSE;
		nStateA_SwitchPress := 0;
	END_IF
	
	IF bPulsePress THEN
		bPulsePress := FALSE;
		nStateA_PulsePress := 0;
	END_IF
	
	IF bPickPut THEN
		bPickPut := FALSE;
		nStateA_PickPut := 0;
	END_IF
	
	nStateA_ResetSpec := 80;
END_IF

SUPER^.A_Reset();
END_ACTION

ACTION A_Stop:
IF nStateA_Stop = 0 THEN

	IF bSetPress THEN
		fbSetPress(bExecute:= FALSE, pPneuChannelRef:= pPneuChannelPress);
	END_IF

	IF bSetVacuum THEN
		fbSetVacuum(bExecute:= FALSE, pPneuChannelRef:= pPneuChannelVac);
	END_IF

	IF bSwitchPress AND nStateA_SwitchPress < 70 THEN
		nStateA_SwitchPress := 70;
	END_IF
	
	IF bPulsePress AND nStateA_PulsePress < 70 THEN
		nStateA_PulsePress := 70;
	END_IF
	
	IF bPickPut AND nStateA_PickPut < 70 THEN
		nStateA_PickPut := 70;
	END_IF

	nStateA_Stop := 1;
END_IF

SUPER^.A_Stop();
END_ACTION

ACTION A_SwitchPress:
// In jedem Zustand sollte umgeschalten werden
CASE nStateA_SwitchPress OF
	0:	//Wie soll geschalten werden?
		IF ePressCtrl = E_PressCtrl.PRESSCTRL_Off THEN
			M_PressAndVacOff();
			eCurrPressCtrl := E_PressCtrl.PRESSCTRL_Off;
			timerPress(IN:= FALSE);
			nStateA_SwitchPress := 80;
			RETURN;
		ELSIF ePressCtrl = E_PressCtrl.PRESSCTRL_PressOn THEN
			M_PressOn();
			eCurrPressCtrl := E_PressCtrl.PRESSCTRL_PressOn;
		ELSIF ePressCtrl = E_PressCtrl.PRESSCTRL_VacOn THEN
			M_VacOn();
			eCurrPressCtrl := E_PressCtrl.PRESSCTRL_VacOn;
		END_IF

		IF tPressTime > T#0MS THEN
			timerPress(IN:= TRUE, PT:= tPressTime);
			nStateA_SwitchPress := 1;
		ELSE
			nStateA_SwitchPress := 80;
		END_IF
		
	1:	//Timer
		//Haben sich die Eingangsparameter geändert?
		IF ePressCtrl <> eCurrPressCtrl THEN
			nStateA_SwitchPress := 0;
			timerPress(IN:= FALSE);
		END_IF
		timerPress();
		IF timerPress.Q THEN
			timerPress(IN:= FALSE);
			M_PressAndVacOff();
			eCurrPressCtrl := E_PressCtrl.PRESSCTRL_Off;
			nStateA_SwitchPress := 80;
		END_IF

	70:	//Abbrechen
		M_PressAndVacOff();
		timerPress(IN:= FALSE);
		nStateA_SwitchPress := 80;
		
	80:	//Haben sich die Eingangsparameter geändert?
		IF ePressCtrl <> eCurrPressCtrl THEN
			nStateA_SwitchPress := 0;
		END_IF
END_CASE
END_ACTION

METHOD FB_init : BOOL
VAR_INPUT
	bInitRetains : BOOL; // if TRUE, the retain variables are initialized (warm start / cold start)
	bInCopyCode : BOOL;  // if TRUE, the instance afterwards gets moved into the copy code (online change)
END_VAR
eObjectType := E_ObjectType.OBJECTTYPE_PickPlacePip;
eObjectGroup := E_ObjectGroup.OBJECTGROUP_MzTool OR E_ObjectGroup.OBJECTGROUP_Device;
END_METHOD

METHOD M_CancelAction
VAR_INPUT
	eAction : E_Action;
END_VAR
CASE eAction OF
	E_Action.ACTION_SetPressure:
		IF bSetPress THEN
			fbSetPress(bExecute:= FALSE, pPneuChannelRef:= pPneuChannelPress);
		END_IF
	
	E_Action.ACTION_SetVacuum:
		IF bSetVacuum THEN
			fbSetVacuum(bExecute:= FALSE, pPneuChannelRef:= pPneuChannelVac);
		END_IF

	E_Action.ACTION_SwitchPressure:
		IF bSwitchPress AND nStateA_SwitchPress < 70 THEN
			nStateA_SwitchPress := 70;
		END_IF

	E_Action.ACTION_PickPutPowder:
		IF bPickPut AND nStateA_PickPut < 70 THEN
			nStateA_PickPut := 70;
		END_IF

	E_Action.ACTION_PulsePressure:
		IF bPulsePress AND nStateA_PulsePress < 70 THEN
			nStateA_PulsePress := 70;
		END_IF	
ELSE
	SUPER^.M_CancelAction(eAction);
END_CASE
END_METHOD

METHOD M_CheckAction : ERRORID
VAR_INPUT
	refActionData 	: REFERENCE TO ST_ActionData;
	pCorrelObject	: POINTER TO FB_Object;
END_VAR

VAR
END_VAR
IF refActionData.eAction = E_Action.ACTION_MeasureTool THEN
	IF fbObjectDirectory.M_GetObjType(refActionData.nTarget) <> E_ObjectType.OBJECTTYPE_TipCalibrator THEN
		M_CheckAction := E_ErrorIdCmd.ERRORID_UnsuitableTarget;
		RETURN;
	END_IF
ELSE
	M_CheckAction := SUPER^.M_CheckAction(refActionData, pCorrelObject);
END_IF
END_METHOD

METHOD M_ExeAction : ERRORID
VAR_INPUT
	refActionData : REFERENCE TO ST_ActionData;	
END_VAR
IF NOT (eCurrentState = E_MachineState.MACHINESTATE_Idle OR
	eCurrentState = E_MachineState.MACHINESTATE_Active OR
	eCurrentState = E_MachineState.MACHINESTATE_Ready) THEN
	M_ExeAction := E_ErrorIdCmd.ERRORID_InvalidState;
	RETURN;
END_IF

CASE refActionData.eAction OF
	
	(*E_Action.ACTION_Init:
		IF NOT bInitAxis AND NOT bInitTool THEN
			bInitAxis := TRUE;
			fbList.A_AddHeadValue( hList := hList, putValue := E_Action.ACTION_Init);	//InitBase
		ELSE
			RETURN;
		END_IF*)		

	E_Action.ACTION_SetPressure:
		fbSetPress(bExecute:= FALSE, pPneuChannelRef:= pPneuChannelPress); //eventueller Fehler wird auch zurückgesetzt
		fbSetPress.bAwait := DINT_TO_BOOL(refActionData.aParams[1]);
		fbSetPress.nValue := DINT_TO_INT(refActionData.aParams[2]);
		fbSetPress.nTolerancePlus := DINT_TO_INT(refActionData.aParams[3]);
		fbSetPress.nToleranceMinus := DINT_TO_INT(refActionData.aParams[4]);
		fbSetPress.tTimeout := DINT_TO_TIME(refActionData.aParams[5]);
		
		fbSetPress(bExecute:= TRUE,	pPneuChannelRef:= pPneuChannelPress,nErrorId=> M_ExeAction);
		IF fbSetPress.bError THEN
			RETURN;
		END_IF
		
		IF NOT bSetPress AND fbSetPress.bBusy THEN
			bSetPress := TRUE;
			fbList.A_AddHeadValue(hList := hList, putValue := E_Action.ACTION_SetPressure);
		ELSE
			RETURN;	
		END_IF

	E_Action.ACTION_SetVacuum:
		fbSetVacuum(bExecute:= FALSE, pPneuChannelRef:= pPneuChannelVac); //eventueller Fehler wird auch zurückgesetzt
		fbSetVacuum.bAwait := DINT_TO_BOOL(refActionData.aParams[1]);
		fbSetVacuum.nValue := DINT_TO_INT(refActionData.aParams[2]);
		fbSetVacuum.nTolerancePlus := DINT_TO_INT(refActionData.aParams[3]);
		fbSetVacuum.nToleranceMinus := DINT_TO_INT(refActionData.aParams[4]);
		fbSetVacuum.tTimeout := DINT_TO_TIME(refActionData.aParams[5]);
		
		fbSetVacuum(bExecute:= TRUE, pPneuChannelRef:= pPneuChannelVac,nErrorId=> M_ExeAction);
		IF fbSetVacuum.bError THEN
			RETURN;
		END_IF
		
		IF NOT bSetVacuum AND fbSetVacuum.bBusy THEN
			bSetVacuum := TRUE;
			fbList.A_AddHeadValue(hList := hList, putValue := E_Action.ACTION_SetVacuum);
		ELSE
			RETURN;	
		END_IF

	E_Action.ACTION_SwitchPressure:
		ePressCtrl := DINT_TO_USINT(refActionData.aParams[1]);
		tPressTime := DINT_TO_TIME(refActionData.aParams[2]);
		IF ePressCtrl = E_PressCtrl.PRESSCTRL_Off OR ePressCtrl = E_PressCtrl.PRESSCTRL_PressOn 
													OR ePressCtrl = E_PressCtrl.PRESSCTRL_VacOn THEN
			IF NOT bSwitchPress THEN
				fbList.A_AddHeadValue(hList := hList, putValue := E_Action.ACTION_SwitchPressure);
				bSwitchPress := TRUE;
			END_IF
		END_IF
				
	E_Action.ACTION_PulsePressure:
		bPulseOn := DINT_TO_BOOL(refActionData.aParams[6]);
		IF bPulseOn THEN	//On
			eSwitchCtrlPhase1 := DINT_TO_USINT(refActionData.aParams[1]);
			eSwitchCtrlPhase2 := DINT_TO_USINT(refActionData.aParams[2]);
	
			IF NOT(refActionData.aParams[4] >= 1 AND refActionData.aParams[4] <= 100) THEN
				M_ExeAction := E_ErrorIdCmd.ERRORID_InvalidDutyCycle;  //Error
				RETURN;
			END_IF
			nTimePhase1 := DINT_TO_UINT(refActionData.aParams[3] / 100 * refActionData.aParams[4]); 
			nTimePhase2 := DINT_TO_UINT(refActionData.aParams[3] - nTimePhase1);
			IF NOT bPulsePress THEN
				bPulsePress := TRUE;
				fbList.A_AddHeadValue(hList := hList, putValue := E_Action.ACTION_PulsePressure);
			ELSE
				RETURN;
			END_IF
			nCurrentPulses := 0;
			nSetpointPulses := DINT_TO_UINT(refActionData.aParams[5]);
		ELSE
			RETURN;
		END_IF				

	E_Action.ACTION_PickPutPowder:
		IF NOT bPickPut THEN
			ePickPutMode := DINT_TO_USINT(refActionData.aParams[1]);
			nIntakeVac := DINT_TO_INT(refActionData.aParams[2]);
			tIntakeTime := DINT_TO_TIME(refActionData.aParams[3]);
			nHoldVac := DINT_TO_INT(refActionData.aParams[4]);
			nBlowOutPress := DINT_TO_INT(refActionData.aParams[5]);
			nBlowOutPulseTime := DINT_TO_UINT(refActionData.aParams[6]);
			nBlowOutPulses := DINT_TO_UINT(refActionData.aParams[7]);
			IF nBlowOutPulseTime = 0 OR nBlowOutPulses = 0 THEN
				RETURN;
			END_IF
			bPickPut := TRUE;
			fbList.A_AddHeadValue(hList := hList, putValue := E_Action.ACTION_PickPutPowder);
		ELSE
			RETURN;	
		END_IF
	ELSE
		M_ExeAction := SUPER^.M_ExeAction(refActionData);
		RETURN;
END_CASE

bBusy := TRUE;
eCurrentState := E_MachineState.MACHINESTATE_Active;
END_METHOD

METHOD M_GetAllProps : ERRORID
VAR_INPUT
	refCmdData : REFERENCE TO  ST_CmdData;
END_VAR
//Basisproperties lesen
SUPER^.M_GetAllProps(refCmdData);
//Specialproperties lesen
nCurrentPropIndex := nCurrentPropIndex + 1; 
IF pPneuChannelPress > 0 THEN
	refCmdData.n32Data[nCurrentPropIndex] := pPneuChannelPress^.nChannel;
ELSE
	refCmdData.n32Data[nCurrentPropIndex] := 0;
END_IF

nCurrentPropIndex := nCurrentPropIndex + 1;
IF pPneuChannelVac > 0 THEN
	refCmdData.n32Data[nCurrentPropIndex] := pPneuChannelVac^.nChannel;
ELSE
	refCmdData.n32Data[nCurrentPropIndex] := 0;
END_IF

nCurrentPropIndex := nCurrentPropIndex + 1;
refCmdData.n32Data[nCurrentPropIndex] := nValveNrPress; //Digitaler Ausgangskanal MzHead Druckventil
nCurrentPropIndex := nCurrentPropIndex + 1;
refCmdData.n32Data[nCurrentPropIndex] := nValveNrVac;	//Digitaler Ausgangskanal MzHead Vakuumventil
END_METHOD

METHOD M_PressAndVacOff
VAR_INPUT
END_VAR
IF nValveNrPress > 0 THEN
	aValves[nValveNrPress].M_Off();
END_IF
IF nValveNrVac > 0 THEN
	aValves[nValveNrVac].M_Off();
END_IF
END_METHOD

METHOD M_PressOn
VAR_INPUT
END_VAR
IF nValveNrPress > 0 THEN
	aValves[nValveNrPress].M_On(1);
END_IF
IF nValveNrVac > 0 THEN
	aValves[nValveNrVac].M_Off();
END_IF
END_METHOD

METHOD M_SetAllProps : ERRORID
VAR_INPUT
	refCmdData : REFERENCE TO  ST_CmdData;
END_VAR

VAR
	nPneuChannel : USINT;
END_VAR
M_SetAllProps := SUPER^.M_SetAllProps(refCmdData);

IF M_SetAllProps > 0 THEN
	RETURN;
END_IF

//PneuChannel Druck
nCurrentPropIndex := nCurrentPropIndex + 1;
nSpecPropIndex := nCurrentPropIndex;
nPneuChannel := DINT_TO_USINT(refCmdData.n32Data[nCurrentPropIndex]);
IF NOT (nPneuChannel > 0 AND nPneuChannel <= cNoOfPneuChannels) THEN
	M_SetAllProps := E_ErrorIdObjMgmt.ERRORID_InvalidPneuChannel;
	RETURN;	
END_IF
pPneuChannelPress := ADR(aFbPneuChannel[nPneuChannel]);

//PneuChannel Vakuum
nCurrentPropIndex := nCurrentPropIndex + 1;
nPneuChannel := DINT_TO_USINT(refCmdData.n32Data[nCurrentPropIndex]);		
IF NOT (nPneuChannel > 0 AND nPneuChannel <= cNoOfPneuChannels) THEN
	M_SetAllProps := E_ErrorIdObjMgmt.ERRORID_InvalidPneuChannel;
	RETURN;	
END_IF
pPneuChannelVac := ADR(aFbPneuChannel[nPneuChannel]);

nCurrentPropIndex := nCurrentPropIndex + 1;
nValveNrPress := DINT_TO_USINT(refCmdData.n32Data[nCurrentPropIndex]); //Digitaler Ausgangskanal MzHead Druckventil Pressure
IF NOT(nValveNrPress >= 0 AND nValveNrPress <= cNoOfValves) THEN
	M_SetAllProps := E_ErrorIdObjMgmt.ERRORID_InvalidMzDOutChannel;
	RETURN;
END_IF

nCurrentPropIndex := nCurrentPropIndex + 1;
nValveNrVac := DINT_TO_USINT(refCmdData.n32Data[nCurrentPropIndex]);	//Digitaler Ausgangskanal MzHead Druckventil Vacuum
IF NOT(nValveNrVac >= 0 AND nValveNrVac <= cNoOfValves) THEN	//kann 0 sein
	M_SetAllProps := E_ErrorIdObjMgmt.ERRORID_InvalidMzDOutChannel;
	RETURN;
END_IF

pZAxisRef^.eFixedToolType := E_MzToolType.TOOL_TYPE_None;

nNoOfProps := nCurrentPropIndex + 1;
END_METHOD

METHOD M_SetSingleProp : ERRORID
VAR_INPUT
	refCmdData : REFERENCE TO  ST_CmdData;
END_VAR

VAR
	nPneuChannel : USINT;
END_VAR
IF nSpecPropIndex = refCmdData.aHeader[1] THEN	//PneuChannel Druck
	nPneuChannel := DINT_TO_USINT(refCmdData.n32Data[0]);
	IF NOT (nPneuChannel > 0 AND nPneuChannel <= cNoOfPneuChannels) THEN
		M_SetSingleProp := E_ErrorIdObjMgmt.ERRORID_InvalidPneuChannel;
		RETURN;	
	END_IF
	pPneuChannelPress := ADR(aFbPneuChannel[nPneuChannel]);
ELSIF (nSpecPropIndex + 1) = refCmdData.aHeader[1] THEN //PneuChannel Vakuum
	nPneuChannel := DINT_TO_USINT(refCmdData.n32Data[0]);
	IF NOT (nPneuChannel >= 0 AND nPneuChannel <= cNoOfPneuChannels) THEN
		M_SetSingleProp := E_ErrorIdObjMgmt.ERRORID_InvalidPneuChannel;
		RETURN;	
	END_IF
	pPneuChannelVac := ADR(aFbPneuChannel[nPneuChannel]);		
ELSIF (nSpecPropIndex + 2) = refCmdData.aHeader[1] THEN
	IF refCmdData.n32Data[0] < 1 OR refCmdData.n32Data[0] > cNoOfValves THEN
		M_SetSingleProp := E_ErrorIdObjMgmt.ERRORID_InvalidValveNumber;
		RETURN;
	END_IF
	nValveNrPress := DINT_TO_USINT(refCmdData.n32Data[0]);	
ELSIF (nSpecPropIndex + 3) = refCmdData.aHeader[1] THEN
	IF refCmdData.n32Data[0] < 1 OR refCmdData.n32Data[0] > cNoOfValves THEN
		M_SetSingleProp := E_ErrorIdObjMgmt.ERRORID_InvalidValveNumber;
		RETURN;
	END_IF
	nValveNrVac := DINT_TO_USINT(refCmdData.n32Data[0]);	
ELSE
	M_SetSingleProp := SUPER^.M_SetSingleProp(refCmdData);
END_IF
END_METHOD

METHOD M_VacOn
VAR_INPUT
END_VAR
IF nValveNrPress > 0 THEN
	aValves[nValveNrPress].M_Off();
END_IF
IF nValveNrVac > 0 THEN
	aValves[nValveNrVac].M_On(1);
END_IF
END_METHOD

END_FUNCTION_BLOCK

// ---- Objects/Targets/Passive/FB_SeptumWaste.TcPOU
FUNCTION_BLOCK FB_SeptumWaste EXTENDS FB_TargetBase
VAR_INPUT
END_VAR
VAR_OUTPUT
END_VAR
VAR
	stWastePoint1	: ST_3DPoint;
	stWastePoint2	: ST_3DPoint;
	nNrOfWastePoints: USINT;
END_VAR

METHOD FB_init : BOOL
VAR_INPUT
	bInitRetains : BOOL; // if TRUE, the retain variables are initialized (warm start / cold start)
	bInCopyCode : BOOL;  // if TRUE, the instance afterwards gets moved into the copy code (online change)
END_VAR
eObjectType := E_ObjectType.OBJECTTYPE_SeptumWaste;
eObjectGroup := E_ObjectGroup.OBJECTGROUP_Target;
END_METHOD

METHOD M_AddChild : ERRORID
VAR_INPUT
	pObject : POINTER TO FB_Object;
	nSlotNr	: UINT;
	nIndex 	: INT;
END_VAR
//Kann folgende Objekte aufnehmen:
//Point, Septum
IF pObject > 0 THEN
	IF pObject^.P_eObjectType = E_ObjectType.OBJECTTYPE_Point OR
		pObject^.P_eObjectType = E_ObjectType.OBJECTTYPE_Septum THEN
		M_AddChild := SUPER^.M_AddChild(pObject,nSlotNr,nIndex);
	ELSE
		M_AddChild := E_ErrorIdObjMgmt.ERRORID_InvalidParentObject;
	END_IF
ELSE
	M_AddChild := E_ErrorIdObjMgmt.ERRORID_InvalidParentObject;
END_IF
END_METHOD

METHOD M_GetAbsPos : ST_3DPoint
VAR_INPUT
	pChildPos	: POINTER TO ST_3DPoint;
	eTargetRef 	: E_TargetRef;
	nParam1		: UINT;
 	nParam2		: UINT;
	nParam3		: USINT;
	nParam4		: USINT;
	nZLevel		: USINT;
END_VAR
VAR_OUTPUT
	nErrorId 	: ERRORID;
	lrAngle		: LREAL;
END_VAR
VAR
	stLocPosLB : ST_3DPoint;
END_VAR
IF eTargetRef = E_TargetRef.TARGETREF_SpecPoint THEN
	stLocPosLB := P_stRelPosLB;
	IF nParam1 = 1 THEN
		stLocPosLB := F_Add3DPoints(stLocPosLB,stWastePoint1);
	ELSIF nParam1 = 2 THEN
		stLocPosLB := F_Add3DPoints(stLocPosLB,stWastePoint2);
	ELSE
		nErrorId := E_ErrorIdCmd.ERRORID_InvalidTargetPointNr;
		RETURN;
	END_IF
	M_GetAbsPos := pParentTarget^.M_GetAbsPos(pChildPos := ADR(stLocPosLB), eTargetRef:= E_TargetRef.TARGETREF_LeftBottom,
												nParam1:= 0,
												nParam2:= 0, nParam3:= 0,nParam4:= 0, nZLevel:= 0,
												lrAngle => lrAngle, nErrorId=> nErrorId);
ELSE
	M_GetAbsPos := SUPER^.M_GetAbsPos(pChildPos := pChildPos, eTargetRef:= eTargetRef,
													nParam1:= nParam1,
													nParam2:= nParam2, nParam3:= nParam3, nParam4:= 0, nZLevel:= nZLevel,
													lrAngle => lrAngle, nErrorId=> nErrorId);
END_IF
END_METHOD

METHOD M_GetAllProps : ERRORID
VAR_INPUT
	refCmdData : REFERENCE TO  ST_CmdData;
END_VAR

VAR
END_VAR
SUPER^.M_GetAllProps(refCmdData); 

nCurrentPropIndex := nCurrentPropIndex + 1;
refCmdData.n32Data[nCurrentPropIndex] := nNrOfWastePoints;
nCurrentPropIndex := nCurrentPropIndex + 1;
refCmdData.n32Data[nCurrentPropIndex] := REAL_TO_DINT(stWastePoint1.X);
nCurrentPropIndex := nCurrentPropIndex + 1;
refCmdData.n32Data[nCurrentPropIndex] := REAL_TO_DINT(stWastePoint1.Y);
nCurrentPropIndex := nCurrentPropIndex + 1;
refCmdData.n32Data[nCurrentPropIndex] := REAL_TO_DINT(stWastePoint1.Z);
nCurrentPropIndex := nCurrentPropIndex + 1;
refCmdData.n32Data[nCurrentPropIndex] := REAL_TO_DINT(stWastePoint2.X);
nCurrentPropIndex := nCurrentPropIndex + 1;
refCmdData.n32Data[nCurrentPropIndex] := REAL_TO_DINT(stWastePoint2.Y);
nCurrentPropIndex := nCurrentPropIndex + 1;
refCmdData.n32Data[nCurrentPropIndex] := REAL_TO_DINT(stWastePoint2.Z);
END_METHOD

METHOD M_SetAllProps : ERRORID
VAR_INPUT
	refCmdData : REFERENCE TO  ST_CmdData;
END_VAR

VAR
END_VAR
M_SetAllProps := SUPER^.M_SetAllProps(refCmdData);

IF M_SetAllProps > 0 THEN
	RETURN;
END_IF

nCurrentPropIndex := nCurrentPropIndex + 1;
//In Abhängigkeit von der Anzahl der Waschpunkte , diese in WastePoints schreiben
nNrOfWastePoints := DINT_TO_USINT(refCmdData.n32Data[nCurrentPropIndex]);
IF NOT (nNrOfWastePoints > 0 AND nNrOfWastePoints <= 2) THEN
	M_SetAllProps := E_ErrorIdObjMgmt.ERRORID_InvalidNoOfSpecPoints;
	RETURN;
END_IF

nCurrentPropIndex := nCurrentPropIndex + 1;
nSpecPropIndex := nCurrentPropIndex;
stWastePoint1.X := DINT_TO_REAL(refCmdData.n32Data[nCurrentPropIndex]);
nCurrentPropIndex := nCurrentPropIndex + 1;
stWastePoint1.Y := DINT_TO_REAL(refCmdData.n32Data[nCurrentPropIndex]);
nCurrentPropIndex := nCurrentPropIndex + 1;
stWastePoint1.Z := DINT_TO_REAL(refCmdData.n32Data[nCurrentPropIndex]);
IF nNrOfWastePoints = 2 THEN
	nCurrentPropIndex := nCurrentPropIndex + 1;
	stWastePoint2.X := DINT_TO_REAL(refCmdData.n32Data[nCurrentPropIndex]);
	nCurrentPropIndex := nCurrentPropIndex + 1;
	stWastePoint2.Y := DINT_TO_REAL(refCmdData.n32Data[nCurrentPropIndex]);
	nCurrentPropIndex := nCurrentPropIndex + 1;
	stWastePoint2.Z := DINT_TO_REAL(refCmdData.n32Data[nCurrentPropIndex]);	
END_IF

nNoOfProps := nCurrentPropIndex + 1;
END_METHOD

METHOD M_SetSingleProp : ERRORID
VAR_INPUT
	refCmdData : REFERENCE TO  ST_CmdData;
END_VAR
IF nSpecPropIndex = refCmdData.aHeader[1] THEN
	stWastePoint1.X := DINT_TO_REAL(refCmdData.n32Data[0]);
ELSIF (nSpecPropIndex + 1) = refCmdData.aHeader[1] THEN
	stWastePoint1.Y := DINT_TO_REAL(refCmdData.n32Data[0]);
ELSIF (nSpecPropIndex + 2) = refCmdData.aHeader[1] THEN
	stWastePoint1.Z := DINT_TO_REAL(refCmdData.n32Data[0]);
ELSIF (nSpecPropIndex + 3) = refCmdData.aHeader[1] THEN
	stWastePoint2.X := DINT_TO_REAL(refCmdData.n32Data[0]);
ELSIF (nSpecPropIndex + 4) = refCmdData.aHeader[1] THEN
	stWastePoint2.Y := DINT_TO_REAL(refCmdData.n32Data[0]);
ELSIF (nSpecPropIndex + 5) = refCmdData.aHeader[1] THEN
	stWastePoint2.Z := DINT_TO_REAL(refCmdData.n32Data[0]);
ELSE
	M_SetSingleProp := SUPER^.M_SetSingleProp(refCmdData);
END_IF
END_METHOD

END_FUNCTION_BLOCK

// ---- Objects/Targets/Passive/FB_SpotPattern.TcPOU
{attribute 'enable_dynamic_creation'}
FUNCTION_BLOCK FB_SpotPattern EXTENDS FB_TargetBase
VAR_INPUT
END_VAR
VAR_OUTPUT
END_VAR
VAR
	nType			: USINT;		//0=TwoDimArray, 1=File
	nCols			: USINT;		//Anzahl Spalten
	nRows			: USINT;		//Anzahl Zeilen
	rSpaceCols		: REAL;			//Abstand Spalten zueinander (Mitte Wells)
	rSpaceRows		: REAL;			//Abstand Zeilen zueinander (Mitte Wells)
	nCurrentCol		: UINT;			//Aktuelle Spalte (nur bei Type "Array")
	nCurrentRow		: UINT;			//Aktuelle Zeile (nur bei Type "Array")
	nCurrentPoint	: UINT;			//Aktueller Punkt (nur bei Type "File")
END_VAR

METHOD FB_init : BOOL
VAR_INPUT
	bInitRetains : BOOL; // if TRUE, the retain variables are initialized (warm start / cold start)
	bInCopyCode : BOOL;  // if TRUE, the instance afterwards gets moved into the copy code (online change)
END_VAR
eObjectType := E_ObjectType.OBJECTTYPE_SpotPattern;
eObjectGroup := E_ObjectGroup.OBJECTGROUP_Target;
END_METHOD

METHOD M_AddChild : ERRORID
VAR_INPUT
	pObject : POINTER TO FB_Object;
	nSlotNr	: UINT;
	nIndex 	: INT;
END_VAR
//Kann folgende Objekte aufnehmen:
IF pObject > 0 THEN
	IF pObject^.P_eObjectType = E_ObjectType.OBJECTTYPE_Point THEN
		M_AddChild := SUPER^.M_AddChild(pObject,nSlotNr,nIndex);
	ELSE
		M_AddChild := E_ErrorIdObjMgmt.ERRORID_InvalidParentObject;
	END_IF
ELSE
	M_AddChild := E_ErrorIdObjMgmt.ERRORID_InvalidParentObject;
END_IF
END_METHOD

METHOD M_GetAllProps : ERRORID
VAR_INPUT
	refCmdData : REFERENCE TO  ST_CmdData;
END_VAR
SUPER^.M_GetAllProps(refCmdData);

nCurrentPropIndex := nCurrentPropIndex + 1;
refCmdData.n32Data[nCurrentPropIndex] := nType;
nCurrentPropIndex := nCurrentPropIndex + 1;
refCmdData.n32Data[nCurrentPropIndex] := nCols;
nCurrentPropIndex := nCurrentPropIndex + 1;
refCmdData.n32Data[nCurrentPropIndex] := nRows;
nCurrentPropIndex := nCurrentPropIndex + 1;
refCmdData.n32Data[nCurrentPropIndex] := REAL_TO_DINT(rSpaceCols);
nCurrentPropIndex := nCurrentPropIndex + 1;
refCmdData.n32Data[nCurrentPropIndex] := REAL_TO_DINT(rSpaceRows);
END_METHOD

METHOD M_SetAllProps : ERRORID
VAR_INPUT
	refCmdData : REFERENCE TO  ST_CmdData;
END_VAR
M_SetAllProps := SUPER^.M_SetAllProps(refCmdData);

IF M_SetAllProps > 0 THEN
	RETURN;
END_IF

nCurrentPropIndex := nCurrentPropIndex + 1;
nType := DINT_TO_USINT(refCmdData.n32Data[nCurrentPropIndex]);
nCurrentPropIndex := nCurrentPropIndex + 1;
nCols := DINT_TO_USINT(refCmdData.n32Data[nCurrentPropIndex]);
nCurrentPropIndex := nCurrentPropIndex + 1; 
nRows := DINT_TO_USINT(refCmdData.n32Data[nCurrentPropIndex]);
nCurrentPropIndex := nCurrentPropIndex + 1;
rSpaceCols := DINT_TO_REAL(refCmdData.n32Data[nCurrentPropIndex]);
nCurrentPropIndex := nCurrentPropIndex + 1;
rSpaceRows := DINT_TO_REAL(refCmdData.n32Data[nCurrentPropIndex]);

nNoOfProps := nCurrentPropIndex + 1;
END_METHOD

METHOD M_SetNextCol : BOOL
VAR_INPUT
END_VAR
nCurrentCol := nCurrentCol + 1;
IF nCurrentCol > nCols THEN //Spaltenumbruch
	nCurrentCol := 1;
	M_SetNextCol := TRUE;
END_IF
END_METHOD

METHOD M_SetNextRow : BOOL
VAR_INPUT
END_VAR
nCurrentRow := nCurrentRow + 1;
IF nCurrentRow > nRows THEN //Zeilenumbruch
	nCurrentRow := 1;
	M_SetNextRow := TRUE;
END_IF
END_METHOD

METHOD M_SetSingleProp : ERRORID
VAR_INPUT
	refCmdData : REFERENCE TO  ST_CmdData;
END_VAR
//Properties Nr kleiner 9 sind Basisproperties
//Dort wird separat auf ihr Gültigkeit geprüft
IF refCmdData.aHeader[1] < 9 THEN	//Property-Nr
	//Basisproperty -> Methode in BasisFb aufrufen
	M_SetSingleProp := SUPER^.M_SetSingleProp(refCmdData);
ELSE	//Specialproperty (ab 9)
	CASE refCmdData.aHeader[1] OF
		9:	nType := DINT_TO_USINT(refCmdData.n32Data[0]);
		
		10:	nCols := DINT_TO_USINT(refCmdData.n32Data[0]);

		11:	nRows := DINT_TO_USINT(refCmdData.n32Data[0]);

		12:	rSpaceCols := DINT_TO_REAL(refCmdData.n32Data[0]);
		
		13:	rSpaceRows := DINT_TO_REAL(refCmdData.n32Data[0]);
		
		ELSE
			//Ungültige Property-Nr
			M_SetSingleProp := E_ErrorIdCmd.ERRORID_InvalidProperty;
	END_CASE
END_IF
END_METHOD

PROPERTY P_nCols : USINT
GET
P_nCols := nCols;
END_GET
END_PROPERTY

PROPERTY P_nRows : USINT
GET
P_nRows := nRows;
END_GET
END_PROPERTY

END_FUNCTION_BLOCK

// ---- Objects/Targets/Passive/FB_NeedleRack.TcPOU
FUNCTION_BLOCK FB_NeedleRack EXTENDS FB_Rack

VAR
	stWasteOffset1 : ST_3DPoint;
	stWasteOffset2 : ST_3DPoint;
END_VAR

METHOD FB_init : BOOL
VAR_INPUT
	bInitRetains : BOOL; // if TRUE, the retain variables are initialized (warm start / cold start)
	bInCopyCode : BOOL;  // if TRUE, the instance afterwards gets moved into the copy code (online change)
END_VAR
eObjectType := E_ObjectType.OBJECTTYPE_NeedleRack;
eObjectGroup := E_ObjectGroup.OBJECTGROUP_Target OR E_ObjectGroup.OBJECTGROUP_Rack;
END_METHOD

METHOD M_AddChild : ERRORID
VAR_INPUT
	pObject : POINTER TO FB_Object;
	nSlotNr	: UINT;	
	nIndex 	: INT;
END_VAR
//Kann folgende Objekte aufnehmen:
//Point, Needles
IF pObject > 0 THEN
	IF pObject^.P_eObjectType = E_ObjectType.OBJECTTYPE_Point THEN
		M_AddChild := SUPER^.M_AddChild(pObject,nSlotNr,nIndex);
	ELSIF pObject^.P_eObjectType = E_ObjectType.OBJECTTYPE_Needle THEN
		//darf nur in ein Slot
		IF nSlotNr > 0 THEN
			M_AddChild := SUPER^.M_AddChild(pObject,nSlotNr,nIndex);
		ELSE
			M_AddChild := E_ErrorIdObjMgmt.ERRORID_InvalidSlotNumber;	
		END_IF
	ELSE
		M_AddChild := E_ErrorIdObjMgmt.ERRORID_InvalidParentObject;
	END_IF
ELSE
	M_AddChild := E_ErrorIdObjMgmt.ERRORID_InvalidParentObject;
END_IF
END_METHOD

METHOD M_CheckAction : ERRORID
VAR_INPUT
	refActionData 	: REFERENCE TO ST_ActionData;
	pCorrelObject	: POINTER TO FB_Object;
END_VAR

VAR
	pSlot 			: POINTER TO FB_PieceSlot;
	pMzTool 		: POINTER TO FB_MzTool;
	pFbUsingPiese 	: POINTER TO FB_UsingPiece;
END_VAR
IF refActionData.eAction = E_Action.ACTION_ExchangePiece THEN
	pSlot := super^.M_GetSlot(DINT_TO_UINT(refActionData.aParams[1]));
	IF pSlot = 0 THEN
		M_CheckAction := E_ErrorIdCmd.ERRORID_InvalidTargetSlot;
	ELSE
		IF refActionData.aParams[2] = 0 THEN //Drop - es darf kein Piece im Slot sein
			IF pSlot^.P_pPiece > 0 THEN
				M_CheckAction := E_ErrorIdCmd.ERRORID_PieceAlreadyInSlot;
				RETURN;	
			END_IF
			pMzTool := fbObjectDirectory.M_GetObjPointer(refActionData.nObject);
			IF pMzTool^.P_pPiece^.P_eObjectType <> E_ObjectType.OBJECTTYPE_Needle THEN
				M_CheckAction := E_ErrorIdCmd.ERRORID_InvalidPieceType;
			END_IF
		ELSIF refActionData.aParams[2] = 1 THEN //Take - es muss ein Piece im Slot
			IF pSlot^.P_pPiece = 0 THEN
				M_CheckAction := E_ErrorIdCmd.ERRORID_NoPieceInSlot;
			ELSE	
				pFbUsingPiese := pSlot^.P_pPiece;
				IF pFbUsingPiese^.P_bUsed THEN
					M_CheckAction := E_ErrorIdCmd.ERRORID_PieceAlreadyUsed;
				END_IF
			END_IF
		ELSE
			M_CheckAction := E_ErrorIdCmd.ERRORID_InvalidCtrl;
		END_IF		
	END_IF
ELSE
	M_CheckAction := SUPER^.M_CheckAction(refActionData, pCorrelObject);
END_IF
END_METHOD

METHOD M_GetAllProps : ERRORID
VAR_INPUT
	refCmdData : REFERENCE TO  ST_CmdData;
END_VAR

VAR
END_VAR
SUPER^.M_GetAllProps(refCmdData);

//WasteOffsets
nCurrentPropIndex := nCurrentPropIndex + 1;
refCmdData.n32Data[nCurrentPropIndex] := REAL_TO_DINT(stWasteOffset1.X);
nCurrentPropIndex := nCurrentPropIndex + 1;
refCmdData.n32Data[nCurrentPropIndex] := REAL_TO_DINT(stWasteOffset1.Y);
nCurrentPropIndex := nCurrentPropIndex + 1;
refCmdData.n32Data[nCurrentPropIndex] := REAL_TO_DINT(stWasteOffset1.Z);
nCurrentPropIndex := nCurrentPropIndex + 1;
refCmdData.n32Data[nCurrentPropIndex] := REAL_TO_DINT(stWasteOffset2.X);
nCurrentPropIndex := nCurrentPropIndex + 1;
refCmdData.n32Data[nCurrentPropIndex] := REAL_TO_DINT(stWasteOffset2.Y);
nCurrentPropIndex := nCurrentPropIndex + 1;
refCmdData.n32Data[nCurrentPropIndex] := REAL_TO_DINT(stWasteOffset2.Z);
END_METHOD

METHOD M_SetAllProps : ERRORID
VAR_INPUT
	refCmdData : REFERENCE TO  ST_CmdData;
END_VAR

VAR
END_VAR
M_SetAllProps := SUPER^.M_SetAllProps(refCmdData);

IF M_SetAllProps > 0 THEN
	RETURN;
END_IF

//WasteOffsets
nCurrentPropIndex := nCurrentPropIndex + 1;
nSpecPropIndex := nCurrentPropIndex;
stWasteOffset1.X := DINT_TO_REAL(refCmdData.n32Data[nCurrentPropIndex]);
nCurrentPropIndex := nCurrentPropIndex + 1;
stWasteOffset1.Y := DINT_TO_REAL(refCmdData.n32Data[nCurrentPropIndex]);
nCurrentPropIndex := nCurrentPropIndex + 1;
stWasteOffset1.Z := DINT_TO_REAL(refCmdData.n32Data[nCurrentPropIndex]);
nCurrentPropIndex := nCurrentPropIndex + 1;
stWasteOffset2.X := DINT_TO_REAL(refCmdData.n32Data[nCurrentPropIndex]);
nCurrentPropIndex := nCurrentPropIndex + 1;
stWasteOffset2.Y := DINT_TO_REAL(refCmdData.n32Data[nCurrentPropIndex]);
nCurrentPropIndex := nCurrentPropIndex + 1;
stWasteOffset2.Z := DINT_TO_REAL(refCmdData.n32Data[nCurrentPropIndex]);
nNoOfProps := nCurrentPropIndex + 1;
END_METHOD

METHOD M_SetSingleProp : ERRORID
VAR_INPUT
	refCmdData : REFERENCE TO  ST_CmdData;
END_VAR
IF nSpecPropIndex = refCmdData.aHeader[1] THEN
	stWasteOffset1.X := DINT_TO_REAL(refCmdData.n32Data[0]);
ELSIF (nSpecPropIndex + 1) = refCmdData.aHeader[1] THEN
	stWasteOffset1.Y := DINT_TO_REAL(refCmdData.n32Data[0]);
ELSIF (nSpecPropIndex + 2) = refCmdData.aHeader[1] THEN
	stWasteOffset1.Z := DINT_TO_REAL(refCmdData.n32Data[0]);
ELSIF (nSpecPropIndex + 3) = refCmdData.aHeader[1] THEN
	stWasteOffset2.X := DINT_TO_REAL(refCmdData.n32Data[0]);
ELSIF (nSpecPropIndex + 4) = refCmdData.aHeader[1] THEN
	stWasteOffset2.Y := DINT_TO_REAL(refCmdData.n32Data[0]);
ELSIF (nSpecPropIndex + 5) = refCmdData.aHeader[1] THEN
	stWasteOffset2.Z := DINT_TO_REAL(refCmdData.n32Data[0]);
ELSE
	M_SetSingleProp := SUPER^.M_SetSingleProp(refCmdData);
END_IF
END_METHOD

PROPERTY P_stWasteOffset1 : ST_3DPoint
GET
P_stWasteOffset1 := stWasteOffset1;
END_GET
END_PROPERTY

PROPERTY P_stWasteOffset2 : ST_3DPoint
GET
P_stWasteOffset2 := stWasteOffset2;
END_GET
END_PROPERTY

END_FUNCTION_BLOCK

// ---- Objects/Targets/Passive/FB_TipRack.TcPOU
FUNCTION_BLOCK FB_TipRack EXTENDS FB_Rack

VAR
END_VAR

METHOD FB_init : BOOL
VAR_INPUT
	bInitRetains : BOOL; // if TRUE, the retain variables are initialized (warm start / cold start)
	bInCopyCode : BOOL;  // if TRUE, the instance afterwards gets moved into the copy code (online change)
END_VAR
eObjectType := E_ObjectType.OBJECTTYPE_TipRack;
eObjectGroup := E_ObjectGroup.OBJECTGROUP_Target OR E_ObjectGroup.OBJECTGROUP_Rack;
END_METHOD

METHOD M_AddChild : ERRORID
VAR_INPUT
	pObject : POINTER TO FB_Object;
	nSlotNr	: UINT;
	nIndex 	: INT;
END_VAR
//Kann folgende Objekte aufnehmen:
//Point, Tips
IF pObject > 0 THEN
	IF pObject^.P_eObjectType = E_ObjectType.OBJECTTYPE_Point THEN
		M_AddChild := SUPER^.M_AddChild(pObject,nSlotNr,nIndex);
	ELSIF pObject^.P_eObjectType = E_ObjectType.OBJECTTYPE_Tip THEN
		//darf nur in ein Slot
		IF nSlotNr > 0 THEN
			M_AddChild := SUPER^.M_AddChild(pObject,nSlotNr,nIndex);
		ELSE
			M_AddChild := E_ErrorIdObjMgmt.ERRORID_InvalidSlotNumber;	
		END_IF
	ELSE
		M_AddChild := E_ErrorIdObjMgmt.ERRORID_InvalidParentObject;
	END_IF
ELSE
	M_AddChild := E_ErrorIdObjMgmt.ERRORID_InvalidParentObject;
END_IF
END_METHOD

METHOD M_CheckAction : ERRORID
VAR_INPUT
	refActionData 	: REFERENCE TO ST_ActionData;
	pCorrelObject	: POINTER TO FB_Object;
END_VAR

VAR
	pSlot : POINTER TO FB_PieceSlot;
	pMzTool : POINTER TO FB_MzTool;
END_VAR
IF refActionData.eAction = E_Action.ACTION_ExchangePiece THEN
	pSlot := super^.M_GetSlot(DINT_TO_UINT(refActionData.aParams[1]));
	IF pSlot = 0 THEN
		M_CheckAction := E_ErrorIdCmd.ERRORID_InvalidTargetSlot;
	ELSE
		IF refActionData.aParams[2] = 0 THEN //Drop - es darf kein Piece im Slot sein
			IF pSlot^.P_pPiece > 0 THEN
				M_CheckAction := E_ErrorIdCmd.ERRORID_PieceAlreadyInSlot;	
				RETURN;
			END_IF
			pMzTool := fbObjectDirectory.M_GetObjPointer(refActionData.nObject);
			IF pMzTool^.P_pPiece^.P_eObjectType <> E_ObjectType.OBJECTTYPE_Tip THEN
				M_CheckAction := E_ErrorIdCmd.ERRORID_InvalidPieceType;
			END_IF			
		ELSIF refActionData.aParams[2] = 1 THEN //Take - es muss ein Piece im Slot
			IF pSlot^.P_pPiece = 0 THEN
				M_CheckAction := E_ErrorIdCmd.ERRORID_NoPieceInSlot;	
			END_IF
		ELSE
			M_CheckAction := E_ErrorIdCmd.ERRORID_InvalidCtrl;	
		END_IF		
	END_IF
ELSE
	M_CheckAction := SUPER^.M_CheckAction(refActionData, pCorrelObject);
END_IF
END_METHOD

END_FUNCTION_BLOCK

// ---- Objects/Targets/Passive/FB_FlipTubeRack.TcPOU
FUNCTION_BLOCK FB_FlipTubeRack EXTENDS FB_Rack

VAR
	stOpenStartPos : ST_3DPoint;
	nOpenMove1DistZ : DINT;
	nOpenMove2DistZ : DINT;
	nOpenMove3DistY : DINT;
	nOpenMove4DistX : DINT;
	nOpenMove5DistZ : DINT;
	stCloseStartPos : ST_3DPoint;
	nCloseMove1DistX : DINT;
	nCloseMove2DistZ : DINT;
END_VAR

METHOD FB_init : BOOL
VAR_INPUT
	bInitRetains : BOOL; // if TRUE, the retain variables are initialized (warm start / cold start)
	bInCopyCode : BOOL;  // if TRUE, the instance afterwards gets moved into the copy code (online change)
END_VAR
eObjectType := E_ObjectType.OBJECTTYPE_FlipTubeRack;
eObjectGroup := E_ObjectGroup.OBJECTGROUP_Target OR E_ObjectGroup.OBJECTGROUP_Rack;
END_METHOD

METHOD M_AddChild : ERRORID
VAR_INPUT
	pObject	: POINTER TO FB_Object;
	nSlotNr	: UINT;
	nIndex 	: INT;
END_VAR
//Kann folgende Objekte aufnehmen:
//Point, Fliptubes
IF pObject > 0 THEN
	IF pObject^.P_eObjectType = E_ObjectType.OBJECTTYPE_Point THEN
		SUPER^.M_AddChild(pObject,nSlotNr,nIndex);
	ELSIF pObject^.P_eObjectType = E_ObjectType.OBJECTTYPE_FlipTube THEN
		//darf nur in ein Slot
		IF nSlotNr > 0 THEN
			SUPER^.M_AddChild(pObject,nSlotNr,nIndex);
		ELSE
			M_AddChild := E_ErrorIdObjMgmt.ERRORID_InvalidSlotNumber;	
		END_IF
	ELSE
		M_AddChild := E_ErrorIdObjMgmt.ERRORID_InvalidParentObject;
	END_IF
ELSE
	M_AddChild := E_ErrorIdObjMgmt.ERRORID_InvalidParentObject;
END_IF
END_METHOD

METHOD M_CheckAction : ERRORID
VAR_INPUT
	refActionData 	: REFERENCE TO ST_ActionData;
	pCorrelObject	: POINTER TO FB_Object;
END_VAR

VAR
	pSlot : POINTER TO FB_PieceSlot;
	pFlipTube : POINTER TO FB_FlipTube;
	pMzTool : POINTER TO FB_MzTool;
END_VAR
IF refActionData.eAction = E_Action.ACTION_OpenCloseFlipTube THEN
	pSlot := super^.M_GetSlot(DINT_TO_UINT(refActionData.aParams[1]));
	IF pSlot = 0 THEN
		M_CheckAction := E_ErrorIdCmd.ERRORID_InvalidTargetSlot;
	ELSE
		//Check, ob FlipTube in Slot
		pFlipTube := pSlot^.P_pPiece;
		IF pFlipTube = 0 THEN
			M_CheckAction := E_ErrorIdCmd.ERRORID_NoPieceInSlot;
		ELSE
			//Wenn geöffnet werden soll, dann muss FlipTube unbedingt geschlosssen sein
			//anders ist es beim Schließen, hier kann Schließen wiederholt werden, fall FlipTube nicht richtig geschlossen
			IF refActionData.aParams[2] = 0 THEN //Open
				IF pFlipTube^.P_bIsOpen THEN
					M_CheckAction := E_ErrorIdCmd.ERRORID_FlipTubeAlreadyOpen;
				END_IF
			END_IF			
		END_IF
	END_IF
ELSIF refActionData.eAction = E_Action.ACTION_InsertTool THEN
	pSlot := super^.M_GetSlot(DINT_TO_UINT(refActionData.aParams[2]));
	IF pSlot = 0 THEN
		M_CheckAction := E_ErrorIdCmd.ERRORID_InvalidTargetSlot;
	ELSE
		//Check, ob FlipTube in Slot
		pFlipTube := pSlot^.P_pPiece;
		IF pFlipTube = 0 THEN
			M_CheckAction := E_ErrorIdCmd.ERRORID_NoPieceInSlot;
		ELSE
		//Tube muss offen sein
			IF NOT pFlipTube^.P_bIsOpen THEN
				M_CheckAction := E_ErrorIdCmd.ERRORID_FlipTubeNotOpen;
			END_IF
		END_IF
	END_IF
ELSE
	M_CheckAction := SUPER^.M_CheckAction(refActionData, pCorrelObject);
END_IF
END_METHOD

METHOD M_GetAllProps : ERRORID
VAR_INPUT
	refCmdData : REFERENCE TO  ST_CmdData;
END_VAR

VAR
END_VAR
SUPER^.M_GetAllProps(refCmdData);

nCurrentPropIndex := nCurrentPropIndex + 1;
refCmdData.n32Data[nCurrentPropIndex] := REAL_TO_DINT(stOpenStartPos.X);
nCurrentPropIndex := nCurrentPropIndex + 1;
refCmdData.n32Data[nCurrentPropIndex] := REAL_TO_DINT(stOpenStartPos.Y);
nCurrentPropIndex := nCurrentPropIndex + 1;
refCmdData.n32Data[nCurrentPropIndex] := REAL_TO_DINT(stOpenStartPos.Z);
nCurrentPropIndex := nCurrentPropIndex + 1;
refCmdData.n32Data[nCurrentPropIndex] := nOpenMove1DistZ;
nCurrentPropIndex := nCurrentPropIndex + 1;
refCmdData.n32Data[nCurrentPropIndex] := nOpenMove2DistZ;
nCurrentPropIndex := nCurrentPropIndex + 1;
refCmdData.n32Data[nCurrentPropIndex] := nOpenMove3DistY;
nCurrentPropIndex := nCurrentPropIndex + 1;
refCmdData.n32Data[nCurrentPropIndex] := nOpenMove4DistX;
nCurrentPropIndex := nCurrentPropIndex + 1;
refCmdData.n32Data[nCurrentPropIndex] := nOpenMove5DistZ;
nCurrentPropIndex := nCurrentPropIndex + 1;
refCmdData.n32Data[nCurrentPropIndex] := REAL_TO_DINT(stCloseStartPos.X);
nCurrentPropIndex := nCurrentPropIndex + 1;
refCmdData.n32Data[nCurrentPropIndex] := REAL_TO_DINT(stCloseStartPos.Y);
nCurrentPropIndex := nCurrentPropIndex + 1;
refCmdData.n32Data[nCurrentPropIndex] := REAL_TO_DINT(stCloseStartPos.Z);
nCurrentPropIndex := nCurrentPropIndex + 1;
refCmdData.n32Data[nCurrentPropIndex] := nCloseMove1DistX;
nCurrentPropIndex := nCurrentPropIndex + 1;
refCmdData.n32Data[nCurrentPropIndex] := nCloseMove2DistZ;
END_METHOD

METHOD M_SetAllProps : ERRORID
VAR_INPUT
	refCmdData : REFERENCE TO  ST_CmdData;
END_VAR

VAR
END_VAR
M_SetAllProps := SUPER^.M_SetAllProps(refCmdData);

IF M_SetAllProps > 0 THEN
	RETURN;
END_IF

nCurrentPropIndex := nCurrentPropIndex + 1;
nSpecPropIndex := nCurrentPropIndex;
stOpenStartPos.X := DINT_TO_REAL(refCmdData.n32Data[nCurrentPropIndex]);
nCurrentPropIndex := nCurrentPropIndex + 1;
stOpenStartPos.Y := DINT_TO_REAL(refCmdData.n32Data[nCurrentPropIndex]);
nCurrentPropIndex := nCurrentPropIndex + 1;
stOpenStartPos.Z := DINT_TO_REAL(refCmdData.n32Data[nCurrentPropIndex]);
nCurrentPropIndex := nCurrentPropIndex + 1;
nOpenMove1DistZ := refCmdData.n32Data[nCurrentPropIndex];
nCurrentPropIndex := nCurrentPropIndex + 1;
nOpenMove2DistZ := refCmdData.n32Data[nCurrentPropIndex];
nCurrentPropIndex := nCurrentPropIndex + 1;
nOpenMove3DistY := refCmdData.n32Data[nCurrentPropIndex];
nCurrentPropIndex := nCurrentPropIndex + 1;
nOpenMove4DistX := refCmdData.n32Data[nCurrentPropIndex];
nCurrentPropIndex := nCurrentPropIndex + 1;
nOpenMove5DistZ := refCmdData.n32Data[nCurrentPropIndex];
nCurrentPropIndex := nCurrentPropIndex + 1;
stCloseStartPos.X := DINT_TO_REAL(refCmdData.n32Data[nCurrentPropIndex]);
nCurrentPropIndex := nCurrentPropIndex + 1;
stCloseStartPos.Y := DINT_TO_REAL(refCmdData.n32Data[nCurrentPropIndex]);
nCurrentPropIndex := nCurrentPropIndex + 1;
stCloseStartPos.Z := DINT_TO_REAL(refCmdData.n32Data[nCurrentPropIndex]);
nCurrentPropIndex := nCurrentPropIndex + 1;
nCloseMove1DistX := refCmdData.n32Data[nCurrentPropIndex];
nCurrentPropIndex := nCurrentPropIndex + 1;
nCloseMove2DistZ := refCmdData.n32Data[nCurrentPropIndex];
nNoOfProps := nCurrentPropIndex + 1;
END_METHOD

METHOD M_SetSingleProp : ERRORID
VAR_INPUT
	refCmdData : REFERENCE TO  ST_CmdData;
END_VAR
IF nSpecPropIndex = refCmdData.aHeader[1] THEN
	stOpenStartPos.X := DINT_TO_REAL(refCmdData.n32Data[0]);
ELSIF (nSpecPropIndex + 1) = refCmdData.aHeader[1] THEN
	stOpenStartPos.Y := DINT_TO_REAL(refCmdData.n32Data[0]);
ELSIF (nSpecPropIndex + 2) = refCmdData.aHeader[1] THEN
	stOpenStartPos.Z := DINT_TO_REAL(refCmdData.n32Data[0]);
ELSIF (nSpecPropIndex + 3) = refCmdData.aHeader[1] THEN
	nOpenMove1DistZ := refCmdData.n32Data[0];
ELSIF (nSpecPropIndex + 4) = refCmdData.aHeader[1] THEN
	nOpenMove2DistZ := refCmdData.n32Data[0];
ELSIF (nSpecPropIndex + 5) = refCmdData.aHeader[1] THEN
	nOpenMove3DistY := refCmdData.n32Data[0];
ELSIF (nSpecPropIndex + 6) = refCmdData.aHeader[1] THEN
	nOpenMove4DistX := refCmdData.n32Data[0];
ELSIF (nSpecPropIndex + 7) = refCmdData.aHeader[1] THEN
	nOpenMove5DistZ := refCmdData.n32Data[0];
ELSIF (nSpecPropIndex + 8) = refCmdData.aHeader[1] THEN
	stCloseStartPos.X := DINT_TO_REAL(refCmdData.n32Data[0]);
ELSIF (nSpecPropIndex + 9) = refCmdData.aHeader[1] THEN
	stCloseStartPos.Y := DINT_TO_REAL(refCmdData.n32Data[0]);
ELSIF (nSpecPropIndex + 10) = refCmdData.aHeader[1] THEN
	stCloseStartPos.Z := DINT_TO_REAL(refCmdData.n32Data[0]);
ELSIF (nSpecPropIndex + 11) = refCmdData.aHeader[1] THEN
	nCloseMove1DistX := refCmdData.n32Data[0];
ELSIF (nSpecPropIndex + 12) = refCmdData.aHeader[1] THEN
	nCloseMove2DistZ := refCmdData.n32Data[0];
ELSE
	M_SetSingleProp := SUPER^.M_SetSingleProp(refCmdData);
END_IF
END_METHOD

PROPERTY P_nCloseMove1DistX : DINT
GET
P_nCloseMove1DistX := nCloseMove1DistX;
END_GET
END_PROPERTY

PROPERTY P_nCloseMove2DistZ : DINT
GET
P_nCloseMove2DistZ := nCloseMove2DistZ;
END_GET
END_PROPERTY

PROPERTY P_nOpenMove1DistZ : DINT
GET
P_nOpenMove1DistZ := nOpenMove1DistZ;
END_GET
END_PROPERTY

PROPERTY P_nOpenMove2DistZ : DINT
GET
P_nOpenMove2DistZ := nOpenMove2DistZ;
END_GET
END_PROPERTY

PROPERTY P_nOpenMove3DistY : DINT
GET
P_nOpenMove3DistY := nOpenMove3DistY;
END_GET
END_PROPERTY

PROPERTY P_nOpenMove4DistX : DINT
GET
P_nOpenMove4DistX := nOpenMove4DistX;
END_GET
END_PROPERTY

PROPERTY P_nOpenMove5DistZ : DINT
GET
P_nOpenMove5DistZ := nOpenMove5DistZ;
END_GET
END_PROPERTY

PROPERTY P_stCloseStartPos : ST_3DPoint
GET
P_stCloseStartPos := stCloseStartPos;
END_GET
END_PROPERTY

PROPERTY P_stOpenStartPos : ST_3DPoint
GET
P_stOpenStartPos := stOpenStartPos;
END_GET
END_PROPERTY

END_FUNCTION_BLOCK

// ---- Objects/Targets/Passive/FB_SeptumRack.TcPOU
FUNCTION_BLOCK FB_SeptumRack EXTENDS FB_Rack

VAR
END_VAR

METHOD FB_init : BOOL
VAR_INPUT
	bInitRetains : BOOL; // if TRUE, the retain variables are initialized (warm start / cold start)
	bInCopyCode : BOOL;  // if TRUE, the instance afterwards gets moved into the copy code (online change)
END_VAR
eObjectType := E_ObjectType.OBJECTTYPE_SeptumRack;
eObjectGroup := E_ObjectGroup.OBJECTGROUP_Target OR E_ObjectGroup.OBJECTGROUP_Rack;
END_METHOD

METHOD M_AddChild : ERRORID
VAR_INPUT
	pObject : POINTER TO FB_Object;
	nSlotNr	: UINT;
	nIndex 	: INT;
END_VAR
//Kann folgende Objekte aufnehmen:
//Point, Septum
IF pObject > 0 THEN
	IF pObject^.P_eObjectType = E_ObjectType.OBJECTTYPE_Point THEN
		M_AddChild := SUPER^.M_AddChild(pObject,nSlotNr,nIndex);
	ELSIF pObject^.P_eObjectType = E_ObjectType.OBJECTTYPE_Septum THEN
		//darf nur in ein Slot
		IF nSlotNr > 0 THEN
			M_AddChild := SUPER^.M_AddChild(pObject,nSlotNr,nIndex);
		ELSE
			M_AddChild := E_ErrorIdObjMgmt.ERRORID_InvalidSlotNumber;	
		END_IF
	ELSE
		M_AddChild := E_ErrorIdObjMgmt.ERRORID_InvalidParentObject;
	END_IF
ELSE
	M_AddChild := E_ErrorIdObjMgmt.ERRORID_InvalidParentObject;
END_IF
END_METHOD

END_FUNCTION_BLOCK

// ---- Objects/Targets/Passive/FB_PortRack.TcPOU
FUNCTION_BLOCK FB_PortRack EXTENDS FB_Rack

VAR
END_VAR

METHOD FB_init : BOOL
VAR_INPUT
	bInitRetains : BOOL; // if TRUE, the retain variables are initialized (warm start / cold start)
	bInCopyCode : BOOL;  // if TRUE, the instance afterwards gets moved into the copy code (online change)
END_VAR
eObjectType := E_ObjectType.OBJECTTYPE_PortRack;
eObjectGroup := E_ObjectGroup.OBJECTGROUP_Target OR E_ObjectGroup.OBJECTGROUP_Rack;
END_METHOD

METHOD M_AddChild : ERRORID
VAR_INPUT
	pObject : POINTER TO FB_Object;
	nSlotNr	: UINT;
	nIndex 	: INT;
END_VAR
//Kann folgende Objekte aufnehmen:
//Point, Ports
IF pObject > 0 THEN
	IF pObject^.P_eObjectType = E_ObjectType.OBJECTTYPE_Point THEN
		M_AddChild := SUPER^.M_AddChild(pObject,nSlotNr,nIndex);
	ELSIF pObject^.P_eObjectType = E_ObjectType.OBJECTTYPE_Port THEN
		//darf nur in ein Slot
		IF nSlotNr > 0 THEN
			M_AddChild := SUPER^.M_AddChild(pObject,nSlotNr,nIndex);
		ELSE
			M_AddChild := E_ErrorIdObjMgmt.ERRORID_InvalidSlotNumber;	
		END_IF
	ELSE
		M_AddChild := E_ErrorIdObjMgmt.ERRORID_InvalidParentObject;
	END_IF
ELSE
	M_AddChild := E_ErrorIdObjMgmt.ERRORID_InvalidParentObject;
END_IF
END_METHOD

METHOD M_CheckAction : ERRORID
VAR_INPUT
	refActionData 	: REFERENCE TO ST_ActionData;
	pCorrelObject	: POINTER TO FB_Object;
END_VAR

VAR
END_VAR
END_METHOD

END_FUNCTION_BLOCK

// ---- Objects/Targets/Passive/FB_pHElectrodeCapRack.TcPOU
FUNCTION_BLOCK FB_pHElectrodeCapRack EXTENDS FB_Rack

VAR
	stHandingOffset : ST_3DPoint;
END_VAR

METHOD FB_init : BOOL
VAR_INPUT
	bInitRetains : BOOL; // if TRUE, the retain variables are initialized (warm start / cold start)
	bInCopyCode : BOOL;  // if TRUE, the instance afterwards gets moved into the copy code (online change)
END_VAR
eObjectType := E_ObjectType.OBJECTTYPE_pHElectrodeCapRack;
eObjectGroup := E_ObjectGroup.OBJECTGROUP_Target OR E_ObjectGroup.OBJECTGROUP_Rack;
END_METHOD

METHOD M_AddChild : ERRORID
VAR_INPUT
	pObject : POINTER TO FB_Object;
	nSlotNr	: UINT;
	nIndex 	: INT;
END_VAR
//Kann folgende Objekte aufnehmen:
//Point, Needles
IF pObject > 0 THEN
	IF pObject^.P_eObjectType = E_ObjectType.OBJECTTYPE_Point THEN
		M_AddChild := SUPER^.M_AddChild(pObject,nSlotNr,nIndex);
	ELSIF pObject^.P_eObjectType = E_ObjectType.OBJECTTYPE_pHElectrodeCap THEN
		//darf nur in ein Slot
		IF nSlotNr > 0 THEN
			M_AddChild := SUPER^.M_AddChild(pObject,nSlotNr,nIndex);
		ELSE
			M_AddChild := E_ErrorIdObjMgmt.ERRORID_InvalidSlotNumber;	
		END_IF
	ELSE
		M_AddChild := E_ErrorIdObjMgmt.ERRORID_InvalidParentObject;
	END_IF
ELSE
	M_AddChild := E_ErrorIdObjMgmt.ERRORID_InvalidParentObject;
END_IF
END_METHOD

METHOD M_CheckAction : ERRORID
VAR_INPUT
	refActionData 	: REFERENCE TO ST_ActionData;
	pCorrelObject	: POINTER TO FB_Object;
END_VAR

VAR
	pSlot 			: POINTER TO FB_PieceSlot;
END_VAR
IF refActionData.eAction = E_Action.ACTION_ExchangePiece THEN
	pSlot := super^.M_GetSlot(DINT_TO_UINT(refActionData.aParams[1]));
	IF pSlot = 0 THEN
		M_CheckAction := E_ErrorIdCmd.ERRORID_InvalidTargetSlot;
	ELSE
		IF refActionData.aParams[2] = 0 THEN //Drop - es darf kein Stamp im Slot sein
			IF pSlot^.P_pPiece > 0 THEN
				M_CheckAction := E_ErrorIdCmd.ERRORID_PieceAlreadyInSlot;	
			END_IF
		ELSIF refActionData.aParams[2] = 1 THEN //Take - es muss ein Stemple im Slot
			IF pSlot^.P_pPiece = 0 THEN
				M_CheckAction := E_ErrorIdCmd.ERRORID_NoPieceInSlot;	
			END_IF
		ELSE
			M_CheckAction := E_ErrorIdCmd.ERRORID_InvalidCtrl;		
		END_IF		
	END_IF
ELSE
	M_CheckAction := SUPER^.M_CheckAction(refActionData, pCorrelObject);
END_IF
END_METHOD

METHOD M_GetAllProps : ERRORID
VAR_INPUT
	refCmdData : REFERENCE TO  ST_CmdData;
END_VAR

VAR
END_VAR
SUPER^.M_GetAllProps(refCmdData);

//WasteOffsets
nCurrentPropIndex := nCurrentPropIndex + 1;
refCmdData.n32Data[nCurrentPropIndex] := REAL_TO_DINT(stHandingOffset.X);
nCurrentPropIndex := nCurrentPropIndex + 1;
refCmdData.n32Data[nCurrentPropIndex] := REAL_TO_DINT(stHandingOffset.Y);
nCurrentPropIndex := nCurrentPropIndex + 1;
refCmdData.n32Data[nCurrentPropIndex] := REAL_TO_DINT(stHandingOffset.Z);
END_METHOD

METHOD M_SetAllProps : ERRORID
VAR_INPUT
	refCmdData : REFERENCE TO  ST_CmdData;
END_VAR

VAR
END_VAR
M_SetAllProps := SUPER^.M_SetAllProps(refCmdData);

IF M_SetAllProps > 0 THEN
	RETURN;
END_IF

//WasteOffsets
nCurrentPropIndex := nCurrentPropIndex + 1;
nSpecPropIndex := nCurrentPropIndex;
stHandingOffset.X := DINT_TO_REAL(refCmdData.n32Data[nCurrentPropIndex]);
nCurrentPropIndex := nCurrentPropIndex + 1;
stHandingOffset.Y := DINT_TO_REAL(refCmdData.n32Data[nCurrentPropIndex]);
nCurrentPropIndex := nCurrentPropIndex + 1;
stHandingOffset.Z := DINT_TO_REAL(refCmdData.n32Data[nCurrentPropIndex]);
nNoOfProps := nCurrentPropIndex + 1;
END_METHOD

METHOD M_SetSingleProp : ERRORID
VAR_INPUT
	refCmdData : REFERENCE TO  ST_CmdData;
END_VAR
IF nSpecPropIndex = refCmdData.aHeader[1] THEN
	stHandingOffset.X := DINT_TO_REAL(refCmdData.n32Data[0]);
ELSIF (nSpecPropIndex + 1) = refCmdData.aHeader[1] THEN
	stHandingOffset.Y := DINT_TO_REAL(refCmdData.n32Data[0]);
ELSIF (nSpecPropIndex + 2) = refCmdData.aHeader[1] THEN
	stHandingOffset.Z := DINT_TO_REAL(refCmdData.n32Data[0]);
ELSE
	M_SetSingleProp := SUPER^.M_SetSingleProp(refCmdData);
END_IF
END_METHOD

PROPERTY P_stHandingOffset : ST_3DPoint
GET
P_stHandingOffset := stHandingOffset;
END_GET
END_PROPERTY

END_FUNCTION_BLOCK

// ---- Objects/Targets/Passive/FB_TipCleanerGen2.TcPOU
FUNCTION_BLOCK FB_TipCleanerGen2 EXTENDS FB_SlotTarget
VAR
	//Spec-Properties
	stWireCleaningStart 	: ST_3DPoint;
	stWireCleaningEnd 		: ST_2DPoint;
	
		
	stBrushCleaningStart	: ST_3DPoint;
	stBrushCleaningEnd 		: ST_2DPoint;
END_VAR

METHOD FB_init : BOOL
VAR_INPUT
	bInitRetains : BOOL; // if TRUE, the retain variables are initialized (warm start / cold start)
	bInCopyCode : BOOL;  // if TRUE, the instance afterwards gets moved into the copy code (online change)
END_VAR
eObjectType := E_ObjectType.OBJECTTYPE_TipCleanerGen2;
eObjectGroup := E_ObjectGroup.OBJECTGROUP_Target;
END_METHOD

METHOD M_AddChild : ERRORID
VAR_INPUT
	pObject : POINTER TO FB_Object;
	nSlotNr	: UINT;
	nIndex 	: INT;
END_VAR
IF pObject > 0 THEN
	IF pObject^.P_eObjectType = E_ObjectType.OBJECTTYPE_CleaningBrush THEN
		M_AddChild := SUPER^.M_AddChild(pObject,nSlotNr,nIndex);
	ELSE
		M_AddChild := E_ErrorIdObjMgmt.ERRORID_InvalidParentObject;
	END_IF
ELSE
	M_AddChild := E_ErrorIdObjMgmt.ERRORID_InvalidParentObject;
END_IF
END_METHOD

METHOD M_CheckAction : ERRORID
VAR_INPUT
	refActionData 	: REFERENCE TO ST_ActionData;
	pCorrelObject	: POINTER TO FB_Object;
END_VAR

VAR
	pSlot : POINTER TO FB_Slot;
END_VAR
IF refActionData.eAction = E_Action.ACTION_CleanTip THEN
	pSlot := super^.M_GetSlot(DINT_TO_UINT(refActionData.aParams[1]));
	IF pSlot = 0 THEN
		M_CheckAction := E_ErrorIdCmd.ERRORID_InvalidTargetSlot;
	ELSE
		IF pSlot^.P_pChild > 0 THEN
			M_CheckAction := E_ErrorIdCmd.ERRORID_NoPieceInSlot;	
		END_IF
	END_IF
ELSE
	M_CheckAction := SUPER^.M_CheckAction(refActionData, pCorrelObject);
END_IF
END_METHOD

METHOD M_GenerateCleaningPoints
VAR_INPUT
	pSlot 	: POINTER TO FB_Slot;
	pNozzle : POINTER TO FB_Nozzle;
END_VAR

VAR
	dRand			: DRAND;
	lrRandNumber	: LREAL;
	pBrush 			: POINTER TO FB_CleaningBrush;
	rMargin			: REAL;
	stDimension		: ST_3DDimension;
	stPositionTemp	: ST_3DPoint;
	stLeftBottom	: ST_2DPoint;
	stRightTop		: ST_2DPoint;
END_VAR
IF pSlot > 0 AND_THEN pSlot^.P_pChild > 0 AND_THEN pSlot^.P_pChild^.P_eObjectType = E_ObjectType.OBJECTTYPE_CleaningBrush THEN
	pBrush := pSlot^.P_pChild;
	stDimension := pBrush^.P_stDimension;
	rMargin := pBrush^.P_rMargin;
	stPositionTemp := pSlot^.P_stAbsPos;
	stLeftBottom.X := stPositionTemp.X;
	stLeftBottom.Y := stPositionTemp.Y;
	stRightTop.X := stPositionTemp.X + stDimension.Width;
	stRightTop.Y := stPositionTemp.Y + stDimension.Depth;
	stBrushCleaningStart.Z := stPositionTemp.Z + stDimension.Height;
	
	//1. Lange Seite ist X
	IF stDimension.Width >= stDimension.Depth THEN
		//Y-Start und Y-End wird zufällig ermittelt
  		stBrushCleaningStart.X := stLeftBottom.X + rMargin - pNozzle^.P_rMeasureDistance / 2;
		stBrushCleaningEnd.X := stRightTop.X  - rMargin + pNozzle^.P_rMeasureDistance / 2;
		dRand(Seed:= DWORD_TO_INT(timeStamp.dwLowDateTime), Num=>lrRandNumber);
		stBrushCleaningStart.Y := LREAL_TO_REAL(stLeftBottom.Y + rMargin + (stDimension.Depth - rMargin * 2) * lrRandNumber);
		dRand(Num=>lrRandNumber);
		stBrushCleaningEnd.Y := LREAL_TO_REAL(stLeftBottom.Y + rMargin + (stDimension.Depth - rMargin * 2) * lrRandNumber);
	ELSE //Lange Seite ist Y
		//X-Start und X-End wird zufällig ermittelt!
  		stBrushCleaningStart.Y := stLeftBottom.Y + rMargin - pNozzle^.P_rMeasureDistance / 2;
		stBrushCleaningEnd.Y := stRightTop.Y - rMargin + pNozzle^.P_rMeasureDistance / 2;
		dRand(Seed:= DWORD_TO_INT(timeStamp.dwLowDateTime), Num=>lrRandNumber);
		stBrushCleaningStart.X := LREAL_TO_REAL(stLeftBottom.X + rMargin +(stDimension.Width - rMargin * 2) * lrRandNumber);
		dRand(Num=>lrRandNumber);
		stBrushCleaningEnd.X := LREAL_TO_REAL(stLeftBottom.X  + rMargin + (stDimension.Width - rMargin * 2) * lrRandNumber);
	END_IF
END_IF
END_METHOD

METHOD M_GetAbsCleaningPos : DINT
VAR_INPUT
	nPosType : USINT;
END_VAR
VAR
	stPoint : ST_3DPoint;
	nWireOffsetX : DINT;
	nWireOffsetY : DINT;
END_VAR
stPoint := P_stAbsPosLB;

IF stDimension.Width >= stDimension.Depth THEN //1. Lange Seite ist X
	nWireOffsetY := 2000;
ELSE
	nWireOffsetX := 2000;
END_IF


CASE nPosType OF
	0: M_GetAbsCleaningPos := REAL_TO_DINT(stWireCleaningStart.X + stPoint.X) + nWireOffsetX;
	1: M_GetAbsCleaningPos := REAL_TO_DINT(stWireCleaningStart.Y + stPoint.Y) + nWireOffsetY;
	2: M_GetAbsCleaningPos := REAL_TO_DINT(stWireCleaningStart.Z + stPoint.Z);
	3: M_GetAbsCleaningPos := REAL_TO_DINT(stWireCleaningEnd.X + stPoint.X) + nWireOffsetX;
	4: M_GetAbsCleaningPos := REAL_TO_DINT(stWireCleaningEnd.Y + stPoint.Y) + nWireOffsetY;
	5: M_GetAbsCleaningPos := REAL_TO_DINT(stWireCleaningEnd.X + stPoint.X) - nWireOffsetX;
	6: M_GetAbsCleaningPos := REAL_TO_DINT(stWireCleaningEnd.Y + stPoint.Y) - nWireOffsetY;
	7: M_GetAbsCleaningPos := REAL_TO_DINT(stWireCleaningStart.X + stPoint.X) - nWireOffsetX;
	8: M_GetAbsCleaningPos := REAL_TO_DINT(stWireCleaningStart.Y + stPoint.Y) - nWireOffsetY;
	//Bei den BrushCleaningPoints wird die absolute Position des Slots bereits in M_GenerateCleaningPoints verrechnent.
	9: M_GetAbsCleaningPos := REAL_TO_DINT(stBrushCleaningStart.X);
	10: M_GetAbsCleaningPos := REAL_TO_DINT(stBrushCleaningStart.Y);
	11: M_GetAbsCleaningPos := REAL_TO_DINT(stBrushCleaningStart.Z);
	12: M_GetAbsCleaningPos := REAL_TO_DINT(stBrushCleaningEnd.X);
	13: M_GetAbsCleaningPos := REAL_TO_DINT(stBrushCleaningEnd.Y);
END_CASE
END_METHOD

METHOD M_GetAllProps : ERRORID
VAR_INPUT
	refCmdData : REFERENCE TO  ST_CmdData;
END_VAR
SUPER^.M_GetAllProps(refCmdData);
nCurrentPropIndex := nCurrentPropIndex + 1;
refCmdData.n32Data[nCurrentPropIndex] := REAL_TO_DINT(stWireCleaningStart.X); 
nCurrentPropIndex := nCurrentPropIndex + 1;
refCmdData.n32Data[nCurrentPropIndex] := REAL_TO_DINT(stWireCleaningStart.Y);
nCurrentPropIndex := nCurrentPropIndex + 1;
refCmdData.n32Data[nCurrentPropIndex] := REAL_TO_DINT(stWireCleaningStart.Z);
nCurrentPropIndex := nCurrentPropIndex + 1;
refCmdData.n32Data[nCurrentPropIndex] := REAL_TO_DINT(stWireCleaningEnd.X);
nCurrentPropIndex := nCurrentPropIndex + 1;
refCmdData.n32Data[nCurrentPropIndex] := REAL_TO_DINT(stWireCleaningEnd.Y);
END_METHOD

{attribute 'TcRpcEnable'}
METHOD M_GetBrushData : ARRAY[0..7] OF DINT
VAR_INPUT
	nSlotNr : UINT;
END_VAR

VAR
	stPosTemp : ST_3DPoint;
	stDimension : ST_3DDimension;
	pSlot : POINTER TO FB_PieceSlot;
	pBrush : POINTER TO FB_CleaningBrush;
END_VAR
pSlot := M_GetSlot(nSlotNr);
IF pSlot > 0 THEN
	stPosTemp := pSlot^.P_stAbsPos;
	IF pSlot^.P_pChild > 0 THEN
		pBrush := pSlot^.P_pChild;
		stDimension := pBrush^.P_stDimension;
	END_IF
END_IF
M_GetBrushData[0] := REAL_TO_DINT(stPosTemp.X);
M_GetBrushData[1] := REAL_TO_DINT(stPosTemp.Y);
M_GetBrushData[2] := REAL_TO_DINT(stDimension.Width);
M_GetBrushData[3] := REAL_TO_DINT(stDimension.Depth);
M_GetBrushData[4] := REAL_TO_DINT(stBrushCleaningStart.X);
M_GetBrushData[5] := REAL_TO_DINT(stBrushCleaningStart.Y);
M_GetBrushData[6] := REAL_TO_DINT(stBrushCleaningEnd.X);
M_GetBrushData[7] := REAL_TO_DINT(stBrushCleaningEnd.Y);
END_METHOD

METHOD M_SetAllProps : ERRORID
VAR_INPUT
	refCmdData : REFERENCE TO  ST_CmdData;
END_VAR

VAR
END_VAR
M_SetAllProps := SUPER^.M_SetAllProps(refCmdData);

IF M_SetAllProps > 0 THEN
	RETURN;
END_IF

nCurrentPropIndex := nCurrentPropIndex + 1;
nSpecPropIndex := nCurrentPropIndex;
stWireCleaningStart.X := DINT_TO_REAL(refCmdData.n32Data[nCurrentPropIndex]);
nCurrentPropIndex := nCurrentPropIndex + 1;
stWireCleaningStart.Y := DINT_TO_REAL(refCmdData.n32Data[nCurrentPropIndex]);
nCurrentPropIndex := nCurrentPropIndex + 1;
stWireCleaningStart.Z := DINT_TO_REAL(refCmdData.n32Data[nCurrentPropIndex]);
nCurrentPropIndex := nCurrentPropIndex + 1;
stWireCleaningEnd.X := DINT_TO_REAL(refCmdData.n32Data[nCurrentPropIndex]);
nCurrentPropIndex := nCurrentPropIndex + 1;
stWireCleaningEnd.Y := DINT_TO_REAL(refCmdData.n32Data[nCurrentPropIndex]);
nNoOfProps := nCurrentPropIndex + 1;
END_METHOD

METHOD M_SetSingleProp : ERRORID
VAR_INPUT
	refCmdData : REFERENCE TO  ST_CmdData;
END_VAR

VAR
	test : INT;
END_VAR
IF nSpecPropIndex = refCmdData.aHeader[1] THEN
 	stWireCleaningStart.X := DINT_TO_REAL(refCmdData.n32Data[0]);
ELSIF (nSpecPropIndex + 1) = refCmdData.aHeader[1] THEN
	stWireCleaningStart.Y := DINT_TO_REAL(refCmdData.n32Data[0]);
ELSIF (nSpecPropIndex + 2) = refCmdData.aHeader[1] THEN
	stWireCleaningStart.Z := DINT_TO_REAL(refCmdData.n32Data[0]);
ELSIF (nSpecPropIndex + 3) = refCmdData.aHeader[1] THEN
	stWireCleaningEnd.X := DINT_TO_REAL(refCmdData.n32Data[0]);
ELSIF (nSpecPropIndex + 4) = refCmdData.aHeader[1] THEN
	stWireCleaningEnd.Y := DINT_TO_REAL(refCmdData.n32Data[0]);
ELSE
	M_SetSingleProp := SUPER^.M_SetSingleProp(refCmdData);
END_IF
END_METHOD

END_FUNCTION_BLOCK

// ---- Objects/Targets/Active/FB_WashStation.TcPOU
FUNCTION_BLOCK FB_WashStation EXTENDS FB_ActiveTarget
VAR
	bLevelSensor		AT %I* : BOOL;
	
	//Spec-Properties
	nNoOfWashPoints 	: USINT;
	nNoOfRinseChannels 	: USINT;
	nPumpNrWastePump	: USINT;
	nSysLiquidBottle 	: USINT;
	nWasteBottle 		: USINT;
	nValveNrAirShower	: USINT;	
	aStRinseChannels	: ARRAY[1..cMaxRinseChannels] OF ST_RinseChannel;
	aStWashPoints		: ARRAY[1..cMaxWashPoints] OF ST_WashPoint;


	//****************************************Aktionvariablen****************************************************
	
	//Action: "SwitchPump"
	bSwitchPump			: BOOL;
	nStateA_SwitchPump	: USINT;
	nSwitchChannel		: USINT;	//0=WasteChannel, 1,2...RinseChannels
	nPumpNrRinsePump	: USINT;
	bSwitchOn			: BOOL;
	bRinsePumpOn		: BOOL;
	
	//Action: "EmptyFluid"
	bEmptyWaste			: BOOL;
	nStateA_EmptyWaste	: USINT;
	tmrEmptyFluid		: TON;
	
	//Action:	"Rinse"
	bRinse				: BOOL;
	nStateA_Rinse		: USINT;
	nRinseChannel		: USINT;
	bRinseOn			: BOOL;
	tmrRinsePause		: TON;
	tmrRinse			: TON;
	bKeepWastePumpOn	: BOOL;
	nGCodeTargetNr		: UINT;
END_VAR

VAR CONSTANT
	cMaxWashPoints 		: USINT := 6;
	cMaxRinseChannels 	: USINT := 2;
END_VAR

IF bInitFB THEN
	bInitFB := FALSE;
	//Fehlerstruktur vorausfüllen
	stError.ObjectId := nObjectID;
	stError.HardwareGrp := E_HardwareGrp.Nothing;
	stError.POU := E_POU.POU_FB_WashStation;
END_IF

CASE eCurrentState OF
	E_MachineState.MACHINESTATE_Idle:
	//Levelsensor checken
	IF NOT bLevelSensor THEN 	//Leeren
		bEmptyWaste := TRUE;
		bBusy := TRUE;
		eCurrentState := E_MachineState.MACHINESTATE_Active;	
	END_IF

	E_MachineState.MACHINESTATE_Active:
	//BasicActions ausführen
	IF bSwitchPump THEN
		A_SwitchPump();
		IF nStateA_SwitchPump >= 80 THEN
			IF nStateA_SwitchPump >= 99 THEN
				bError := TRUE;	
			END_IF
			bSwitchPump := FALSE;
			nStateA_SwitchPump := 0;
		END_IF
	END_IF
	
	IF bEmptyWaste THEN
		A_EmptyWaste();
		IF nStateA_EmptyWaste >= 80 THEN
			IF nStateA_EmptyWaste >= 99 THEN
				bError := TRUE;	
			END_IF
			bEmptyWaste := FALSE;
			nStateA_EmptyWaste := 0;
		END_IF
	END_IF
	
	IF bRinse THEN
		A_Rinse();
		IF nStateA_Rinse >= 80 THEN
			IF nStateA_Rinse >= 99 THEN
				bError := TRUE;	
			END_IF
			bRinse := FALSE;
			nStateA_Rinse := 0;
		END_IF
	END_IF
	
	IF NOT (bSwitchPump OR bEmptyWaste OR bRinse) THEN
		bBusy := FALSE;
		eCurrentState := E_MachineState.MACHINESTATE_Idle;
	END_IF
	
	E_MachineState.MACHINESTATE_Reset:
		bError := FALSE;
		
END_CASE

